# B&R Automation Studio project SuperTrakProject
Automation Studio 6.7.1.5

## Configuration APC4100

CPU 5APC4100.TGL1-000, AutomationRuntime 6.7.6, Build 11.3.0

### Task classes (Cpu.sw)
```
Cyclic#1 (cycle 800 us, tolerance 0 us):
  STCyclic <- Source.STMgr.STCyclic.STCyclic.prg
  STSystem <- Source.STMgr.STSystem.STSystem.prg
  STSection <- Source.STMgr.STSection.STSection.prg
  STTarget <- Source.STMgr.STTarget.STTarget.prg
  STShuttle <- Source.STMgr.STShuttle.STShuttle.prg
Cyclic#2 (cycle 1600 us, tolerance 1600 us):
  Main <- Source.MachineMgr.Main.prg
Cyclic#3 (cycle 20000 us, tolerance 20000 us):
  EipComm <- Source.EthIP.EipComm.prg
DataObjects: ethIPcon <- Source.EthIP.ethIPcon.dob
Binaries: udbdef, TCData, TCLang, ashwd, ashwac, sysconf, asfw, arconfig, TC, varmap, stcyclicvm
Libraries: ArEventLog, AsIOAcc, AsARCfg, AsArProf, AsArSdm, AsGuard, AsHttp, AsIO, AsIODiag, AsIOMMan, AsIoTime, AsTCP, astime, AsUDP, AsXml, brsystem, DataObj, FileIO, sys_lib, runtime, AsBrStr, standard, AsIecCon, AsEthIP, StCom, SuperTrak, ArTextSys, UserLog, aspciext
```

### Hardware
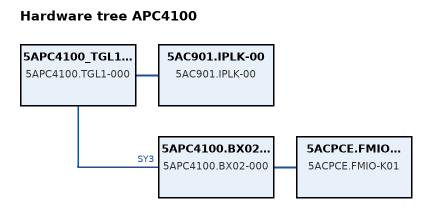
```
5AC901.IPLK-00 : 5AC901.IPLK-00 v2.1.0.0  [SS -> 5APC4100_TGL1_000.SS2]
  Connector IF1:
    CycleTime = 800
5ACPCE.FMIO-K01 : 5ACPCE.FMIO-K01 v1.0.6.0  [SL -> 5APC4100.BX02-000.SL1]
5APC4100.BX02-000 : 5APC4100.BX02-000 v1.0.0.0  [SY -> 5APC4100_TGL1_000.SY3]
5APC4100_TGL1_000 : 5APC4100.TGL1-000 v1.4.0.0
  Connector IF3:
    AssignedOperatingSystem = ARemb
    ActivateDevice = 1
    HostName = apc4100_supertrak
    Mode = Manual
    InternetAddress = 192.168.1.100
    SubnetMask = 255.255.255.0
    ActivateSnmp = 2
  Connector IF4:
    AssignedOperatingSystem = ARemb
    ActivateDevice = 1
    HostName = apc4100_supertrak
    Mode = Manual
    InternetAddress = 10.10.6.10
    SubnetMask = 255.255.255.0
    ActivateSnmp = 2
  Connector IF5:
    AssignedOperatingSystem = ARemb
    ActivateDevice = 1
    HostName = apc4100_supertrak
    ActivateSnmp = 2
  Connector IF6:
    AssignedOperatingSystem = ARemb
    ActivateDevice = 1
    HostName = apc4100_supertrak
    ActivateSnmp = 2
  Connector IF7:
    AssignedOperatingSystem = ARemb
  Connector IF8:
    AssignedOperatingSystem = ARemb
  Connector IF9:
    AssignedOperatingSystem = ARemb
  Connector IF10:
    AssignedOperatingSystem = ARemb
  Connector IF11:
    AssignedOperatingSystem = ARemb
  Connector IF12:
    AssignedOperatingSystem = ARemb
  ConfigurationID = SuperTrakProject_APC4100
  ConfigVersion = 2.0.0
  UserPartitionSize = 100
  EnableDebugger = 1
  TimerDeviceType = EPLX2X
  TimerDevice = 5AC901.IPLK-00.IF1
  TaskClassIdleTime = 800
  Cyclic1Duration = 800
  Cyclic1Tolerance = 0
  Cyclic2Duration = 1600
  Cyclic2Tolerance = 1600
  Cyclic3Duration = 20000
  Cyclic3Tolerance = 20000
  Cyclic8Duration = 9600
  FileDevice1
  FileDeviceName1 = USER
  FileDevicePath1 = USER_PATH
  EthernetHostName = apc4100_supertrak
  ActivateFtpServer = 1
  FtpUser1
  FtpUsername1 = SuperTrakUser
  FtpUserPassword1 = ss9kzLCmIlqrwmUb/fXl5DaWp4kAdzlsqUsPLdKHEtE=  // SuperTrak
  FtpUserSalt1 = yN37R9W0
  FTPAccessRight1 = 0
  ActivateWebServer = 1
  WebServerProtocol = 1
  ActivateSdm = 1
  Authentication = 0
```

## Configuration APC910

CPU 5APC4100.TGL1-000, AutomationRuntime 6.3.4, Build 11.3.0, Vc 6.0.0

CPU 5PC900.TS17-00, AutomationRuntime 6.3.4, Build 11.3.0, Vc 6.0.0

CPU 5PC900.TS77-00, AutomationRuntime G4.91, Build 4.1.2, Vc V4.72.5

### Task classes (Cpu.sw)
```
Cyclic#1 (cycle 800 us, tolerance 0 us):
  STCyclic <- Source.STMgr.STCyclic.STCyclic.prg
  STSystem <- Source.STMgr.STSystem.STSystem.prg [disabled]
  STSection <- Source.STMgr.STSection.STSection.prg [disabled]
  STTarget <- Source.STMgr.STTarget.STTarget.prg [disabled]
  STShuttle <- Source.STMgr.STShuttle.STShuttle.prg [disabled]
Cyclic#2 (cycle 1600 us, tolerance 1600 us):
  Main <- Source.MachineMgr.Main.prg [disabled]
Cyclic#4:
  EipComm <- Source.EthIP.EipComm.prg [disabled]
DataObjects: ethIPcon <- Source.EthIP.ethIPcon.dob
Binaries: STComTexts, udbdef, TCData, TCLang, ashwd, ashwac, sysconf, asfw, arconfig, TC, varmap, stcyclicvm
Libraries: SuperTrak, ArEventLog, AsIOAcc, AsARCfg, AsArLog, AsArProf, AsArSdm, AsGuard, AsHttp, AsIO, AsIODiag, AsIOMMan, AsIoTime, AsTCP, astime, AsUDP, AsXml, brsystem, DataObj, FileIO, sys_lib, runtime, StCom, AsBrStr, standard, AsIecCon, UserLog, AsEthIP, aspciext
```

### Task classes (Cpu.sw)
```
Cyclic#1 (cycle 800 us, tolerance 0 us):
  STCyclic <- Source.STMgr.STCyclic.STCyclic.prg
  STSystem <- Source.STMgr.STSystem.STSystem.prg
  STSection <- Source.STMgr.STSection.STSection.prg
  STTarget <- Source.STMgr.STTarget.STTarget.prg
  STShuttle <- Source.STMgr.STShuttle.STShuttle.prg
Cyclic#2 (cycle 1600 us, tolerance 1600 us):
  Main <- Source.MachineMgr.Main.prg
Cyclic#4:
  EipComm <- Source.EthIP.EipComm.prg
DataObjects: ethIPcon <- Source.EthIP.ethIPcon.dob
Binaries: STComTexts, udbdef, TCData, TCLang, ashwd, ashwac, sysconf, asfw, arconfig, TC, varmap, stcyclicvm
Libraries: SuperTrak, ArEventLog, AsIOAcc, AsARCfg, AsArLog, AsArProf, AsArSdm, AsGuard, AsHttp, AsIO, AsIODiag, AsIOMMan, AsIoTime, AsTCP, astime, AsUDP, AsXml, brsystem, DataObj, FileIO, sys_lib, runtime, StCom, AsBrStr, standard, AsIecCon, UserLog, AsEthIP, aspciext
```

### Hardware
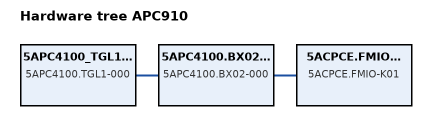
```
5ACPCE.FMIO-K01 : 5ACPCE.FMIO-K01 v1.0.6.0  [SL -> 5APC4100.BX02-000.SL1]
5APC4100.BX02-000 : 5APC4100.BX02-000 v1.0.0.0  [SY -> 5APC4100_TGL1_000.SY3]
5APC4100_TGL1_000 : 5APC4100.TGL1-000 v1.2.0.0
  Connector IF3:
    AssignedOperatingSystem = ARemb
    ActivateDevice = 1
    HostName = apc910_supertrak
    Mode = Manual
    InternetAddress = 192.168.1.100
    SubnetMask = 255.255.255.0
    ActivateSnmp = 2
  Connector IF4:
    AssignedOperatingSystem = ARemb
    ActivateDevice = 1
    HostName = apc910_supertrak
    Mode = Manual
    InternetAddress = 10.10.6.10
    SubnetMask = 255.255.255.0
    ActivateSnmp = 2
  Connector IF5:
    AssignedOperatingSystem = ARemb
    ActivateDevice = 1
  Connector IF6:
    AssignedOperatingSystem = ARemb
    ActivateDevice = 1
  Connector IF7:
    AssignedOperatingSystem = ARemb
  Connector IF8:
    AssignedOperatingSystem = ARemb
  Connector IF9:
    AssignedOperatingSystem = ARemb
  Connector IF10:
    AssignedOperatingSystem = ARemb
  Connector IF11:
    AssignedOperatingSystem = ARemb
  Connector IF12:
    AssignedOperatingSystem = ARemb
  ConfigurationID = SuperTrakProject_APC910
  ConfigVersion = 1.1.0
  UserPartitionSize = 100
  SystemTick = 800
  TaskClassIdleTime = 800
  Cyclic1Duration = 800
  Cyclic1Tolerance = 0
  Cyclic2Duration = 1600
  Cyclic2Tolerance = 1600
  Cyclic3Duration = 49600
  Cyclic3Tolerance = 49600
  Cyclic8Duration = 9600
  FileDevice1
  FileDeviceName1 = USER
  FileDevicePath1 = USER_PATH
  EthernetHostName = apc910_supertrak
  ActivateFtpServer = 1
  FtpUser1
  FtpUsername1 = SuperTrakUser
  FtpUserPassword1 = ss9kzLCmIlqrwmUb/fXl5DaWp4kAdzlsqUsPLdKHEtE=  // SuperTrak
  FtpUserSalt1 = yN37R9W0
  FTPAccessRight1 = 0
  ActivateWebServer = 1
  ActivateSdm = 1
```

### VarMap.vvm - 5PC900_TS17_00/VarMap.vvm
```iecst
VAR_CONFIG
	Cyclic#1.::gSTSection.Cmd AT %Q.Cyclic#1.::STSection:Interface.Cmd;
	Cyclic#1.::STSection:Interface.Status AT %Q.Cyclic#1.::gSTSection.Status;
END_VAR
```

### STCyclicVM.vvm - 5PC900_TS17_00/VariableMap/STCyclicVM.vvm
```iecst
VAR_CONFIG
	::STCyclic:Interface.Status AT %Q.::gSTCyclic.Status;
END_VAR
```

### STSystemVM.vvm - 5PC900_TS17_00/VariableMap/STSystemVM.vvm
```iecst
VAR_CONFIG
	::gSTSystem.Par AT %Q.::STSystem:Interface.Par;
END_VAR
```

### VarMap.vvm - 5PC900_TS77_00/VarMap.vvm
```iecst
VAR_CONFIG
	::gSTSystem.Cmd AT %Q.::STSystem:Interface.Cmd;
	::STSystem:Interface.Status AT %Q.::gSTSystem.Status;
	::gSTSection.Cmd AT %Q.::STSection:Interface.Cmd;
	::gSTSection.Par AT %Q.::STSection:Interface.Par;
	::STSection:Interface.Status AT %Q.::gSTSection.Status;
END_VAR
```

## Logical view

Binary libraries used (declarations not repeated): SuperTrak 0.63.4, StCom 6.0.0, brsystem, runtime, sys_lib, standard, astime, AsBrStr, AsIecCon, AsIOAcc, AsARCfg, AsArProf, AsArSdm, AsGuard, AsHttp, AsIO, AsIODiag, AsIOMMan, AsIoTime, AsTCP, AsUDP, AsXml, DataObj, FileIO, ArEventLog, UserLog 2.1.0, ArTextSys, AsEthIP

### Package Logical/Libraries - Global libraries

### Library Logical/Libraries/StHelper (IEC)
Depends on: SuperTrak, UserLog

#### Constants.var - Exported constants
```iecst
VAR CONSTANT
	ST_HELPER_FUNCTION_INPUT_ERROR : UINT := 20; (*Helper Function could not execute due to an invalid input*)
END_VAR
```

#### StHelper.fun - Exported functions and function blocks
```iecst
(*Data Parameters*)

FUNCTION GetDataParameterArrayLength : UINT (*Gets the array length for data parameters. The array length N indicates that N values can be addressed, using indexes 0 through (N - 1). Returned value is the Status of SuperTrakServChanRead*)
	VAR_INPUT
		ParameterToCheck : UINT; (*Data parameter number to check the length of*)
		pDataBuffer : UDINT; (*Pointer to (UDINT) location of output data*)
		DataBufferLength : UINT; (*[bytes] Size of output data location*)
	END_VAR
	VAR
		LogValues : UserLogFormatType; (*Runtime values formatted for Log messages*)
	END_VAR
END_FUNCTION
(*Inputs and Outputs*)

FUNCTION GetInputFunctions : UINT (*Gets the functions configured for all Trakmaster Inputs. Returned value is the Status of SuperTrakServChanRead*)
	VAR_INPUT
		pDataBuffer : UDINT; (*Pointer to (UINT[8]) location of output data. Each element in the array is a Digital Input.*)
		DataBufferLength : UINT; (*[bytes] Size of output data location*)
	END_VAR
	VAR
		GetArrayLengthStatus : UINT; (*Status returned by GetDataParameterArrayLength*)
		GetArrayLengthReturnValue : UDINT; (*Value returned by GetDataParameterArrayLength*)
		Count : UINT; (*Count of values to read*)
		LogValues : UserLogFormatType; (*Runtime values formatted for Log messages*)
	END_VAR
END_FUNCTION

FUNCTION SetInputFunctions : UINT (*Sets the functions configured for all Trakmaster Inputs. Returned value is the Status of SuperTrakServChanRead*)
	VAR_INPUT
		pDataBuffer : UDINT; (*Pointer to (UINT[8]) location of input data. Each element in the array is a Digital Input.*)
		DataBufferLength : UINT; (*[bytes] Size of input data location*)
	END_VAR
	VAR
		GetArrayLengthStatus : UINT; (*Status returned by GetDataParameterArrayLength*)
		GetArrayLengthReturnValue : UDINT; (*Value returned by GetDataParameterArrayLength*)
		Count : UINT; (*Count of values to read*)
		LogValues : UserLogFormatType; (*Runtime values formatted for Log messages*)
	END_VAR
END_FUNCTION
```

#### GetDataParameterArrayLength.st
```iecst
// Gets the array length for data parameters. The array length N indicates that N values can be addressed, using indexes 0 through (N - 1)
// An array length of 1 indicates that a single value can be addressed at index 0.
// An array length OF 0 indicates that the parameter is NOT available.
// Returned value is the Status of SuperTrakServChanRead
FUNCTION GetDataParameterArrayLength

    IF (ParameterToCheck < 1024) OR (pDataBuffer = 0) OR (DataBufferLength = 0) THEN
        GetDataParameterArrayLength := ST_HELPER_FUNCTION_INPUT_ERROR;
    ELSE
        // Data parameters occupy parameter numbers starting at 1024
        // To obtain information about data parameter K, specify index K - 1024 when reading the Data Parameter Information parameters
        GetDataParameterArrayLength := SuperTrakServChanRead(0, stPAR_PARAM_ARRAY_LENGTH, ParameterToCheck - 1024, 1, pDataBuffer, DataBufferLength);
        LogValues.i[0] := stPAR_PARAM_ARRAY_LENGTH;
        LogValues.i[1] := ParameterToCheck - 1024;
        LogValues.i[2] := 1;
        UserLogAdvanced(USERLOG_SEVERITY_INFORMATION, 100, 'Service Channel Request: Parameter %i, Start Index %i, Count %i', LogValues);
    END_IF;

END_FUNCTION
```

#### InputsAndOutputs.st
```iecst
// Gets the functions configured for all Trakmaster Inputs. Returned value is the Status of SuperTrakServChanRead
FUNCTION GetInputFunctions

    // Check inputs for validity
    IF (pDataBuffer = 0) OR (DataBufferLength = 0) THEN
        GetInputFunctions := ST_HELPER_FUNCTION_INPUT_ERROR;
        RETURN;
    END_IF;

    // Check size of data array
    GetArrayLengthStatus := GetDataParameterArrayLength(stPAR_DIGITAL_INPUT_FUNCTION, ADR(GetArrayLengthReturnValue), SIZEOF(GetArrayLengthReturnValue));
    IF GetArrayLengthStatus <> 0 THEN
        GetInputFunctions := ST_HELPER_FUNCTION_INPUT_ERROR;
        RETURN;
    END_IF;

    // Number of inputs is lesser of (data array size, size of data buffer elements)
    Count := MIN(UDINT_TO_UINT(GetArrayLengthReturnValue), DataBufferLength/SIZEOF(UINT));
    GetInputFunctions := SuperTrakServChanRead(0, stPAR_DIGITAL_INPUT_FUNCTION, 0, Count, pDataBuffer, DataBufferLength);
    LogValues.i[0] := stPAR_DIGITAL_INPUT_FUNCTION;
    LogValues.i[1] := 0;
    LogValues.i[2] := Count;
    UserLogAdvanced(USERLOG_SEVERITY_INFORMATION, 100, 'Service Channel Request: Parameter %i, Start Index %i, Count %i', LogValues);

END_FUNCTION

// Sets the functions configured for all Trakmaster Inputs. Returned value is the Status of SuperTrakServChanRead
FUNCTION SetInputFunctions

    // Check inputs for validity
    IF (pDataBuffer = 0) OR (DataBufferLength = 0) THEN
        SetInputFunctions := ST_HELPER_FUNCTION_INPUT_ERROR;
        RETURN;
    END_IF;

    // Check size of data array
    GetArrayLengthStatus := GetDataParameterArrayLength(stPAR_DIGITAL_INPUT_FUNCTION, ADR(GetArrayLengthReturnValue), SIZEOF(GetArrayLengthReturnValue));
    IF GetArrayLengthStatus <> 0 THEN
        SetInputFunctions := ST_HELPER_FUNCTION_INPUT_ERROR;
        RETURN;
    END_IF;

    // Number of inputs is lesser of (data array size, size of data buffer elements)
    Count := MIN(UDINT_TO_UINT(GetArrayLengthReturnValue), DataBufferLength/SIZEOF(UINT));
    SetInputFunctions := SuperTrakServChanWrite(0, stPAR_DIGITAL_INPUT_FUNCTION, 0, Count, pDataBuffer, DataBufferLength);
    LogValues.i[0] := stPAR_DIGITAL_INPUT_FUNCTION;
    LogValues.i[1] := 0;
    LogValues.i[2] := Count;
    UserLogAdvanced(USERLOG_SEVERITY_INFORMATION, 100, 'Service Channel Request: Parameter %i, Start Index %i, Count %i', LogValues);

END_FUNCTION
```

### Package Logical/Source/MachineMgr - Machine manager

### Machine.typ - Global Machine types
```iecst
(***************************************************************************************
 * Global Machine data types
 *
 * These structures allow any program (task) to interface with the Main Machine task
 *
 * File: Machine.typ
 * Created: 2024-08-15
 *
 * Authors:
 *  Marcus Mangel, B&R Industrial Automation
 *
****************************************************************************************)

TYPE
    Machine_type :     STRUCT  (*Machine interface*)
        Cmd : Machine_Cmd_type; (*Machine commands*)
        Par : Machine_Par_type; (*Machine parameters*)
        Status : Machine_Status_type; (*Machine statuses*)
    END_STRUCT;
    Machine_Cmd_type :     STRUCT  (*Machine commands*)
        Power : BOOL; (*Power all SuperTrak sections*)
        Run : BOOL; (*Run process sequence*)
        ErrorReset : BOOL; (*Error reset*)
    END_STRUCT;
    Machine_Par_type :     STRUCT  (*Machine parameters*)
        Velocity : REAL := 1500.0; (*[mm/s] Set velocity for target and shuttle release commands*)
        Acceleration : REAL := 15.0; (*[m/s^2] Set acceleration for target and shuttle release commands*)
    END_STRUCT;
    Machine_Status_type :     STRUCT  (*Machine statuses*)
        PowerOn : BOOL; (*The main state machine is enabled and the trak is powered*)
        Ready : BOOL; (*The program is ready to run*)
        Error : BOOL; (*There is an active error present*)
        ErrorType : Error_Type_enum; (*Source of the last error*)
        ErrorText : STRING[255];
        SuperTrakDiag : SuperTrak_Diag_type; (*Fault and Warning information from the SuperTrak library*)
    END_STRUCT;
    Error_Type_enum :
        ( (*Source of the last error*)
        errNONE := 0,
        errUSER := 1, (*See Automation Studio code*)
        errST_COM_SYSTEM := 2, (*See documentation for the StCom or SuperTrak libraries in Automation Studio*)
        errST_COM_SECTION := 3, (*See documentation for the StCom or SuperTrak libraries in Automation Studio*)
        errST_SYSTEM := 10, (*See "Faults" section in TrakMaster Help *)
        warnST_SYSTEM := 11, (*See "Warnings" section in TrakMaster Help *)
        errST_SECTION := 20, (*See "Faults" section in TrakMaster Help *)
        warnST_SECTION := 21, (*See "Warnings" section in TrakMaster Help *)
        errST_COM_TARGET := 30, (*See documentation for the StCom or SuperTrak libraries in Automation Studio*)
        errST_COM_SHUTTLE := 40 (*See documentation for the StCom or SuperTrak libraries in Automation Studio*)
        );
    SuperTrak_Diag_type :     STRUCT  (*Fault and Warning information from the SuperTrak library*)
        SuperTrakDiagIndex : USINT; (*Index 0 is the System, others are for a specific section. Set to a relevant index when Errors occur*)
        Warnings : ARRAY[0..31]OF BOOL; (*See TrakMaster Help for descriptions*)
        Errors : ARRAY[0..31]OF BOOL; (*See TrakMaster Help for descriptions*)
    END_STRUCT;
END_TYPE
```

### Machine.var - Global Machine variables
```iecst
(***************************************************************************************
 * Global Machine variables
 *
 * These variables allow any program (task) to interface with the Main Machine task
 *
 * File: Machine.var
 * Created: 2024-08-15
 *
 * Authors:
 *  Marcus Mangel, B&R Industrial Automation
 *
***************************************************************************************)
VAR
    gMachine : Machine_type; (*Machine interface*)
    gUseExternalControl : BOOL;
END_VAR
```

### Program Logical/Source/MachineMgr/Main (IEC) - Main Machine control

#### Main.st - Init, cyclic, exit code
```iecst
(***************************************************************************************
 * Main task
 *
 * This task (program) provides a state machine for controlling any and all hardware
 * connected to the B&R PC. SuperTrak (Target) release code is demonstrated in the
 * MAIN_STATE_RUN (Running) state of this state machine.
 *
 * Other tasks can interface with this one via the global variable "gMachine".
 *
 * File: Main.st
 * Created: 2024-08-15
 *
 * Authors:
 *  Marcus Mangel, B&R Industrial Automation
 *  Bryan Olson, B&R Industrial Automation
 *
***************************************************************************************)

PROGRAM _INIT

    // Set simulated station timer values
    SimulatedProcessTimes[ST_TARGET_LOAD] := T#1s;
    SimulatedProcessTimes[ST_TARGET_QUEUE] := T#100ms;
    SimulatedProcessTimes[ST_TARGET_PROCESS] := T#500ms;
    SimulatedProcessTimes[ST_TARGET_UNLOAD] := T#1s;

END_PROGRAM

PROGRAM _CYCLIC

    // Copy inputs
    Interface.Cmd := gMachine.Cmd;
    Interface.Par := gMachine.Par;

    // Check for command edges
    r_trig_Power(CLK := Interface.Cmd.Power);
    r_trig_Run(CLK := Interface.Cmd.Run);

    // Translate Errors
    GetErrorType;
    GetTrakMasterWarningsAndErrors;
    // Catch SuperTrak Errors
    IF gSuperTrak.System.Status.Error OR gSuperTrak.System.Info.FaultPresent
        OR gSuperTrak.Sections.Status.Error OR (gSuperTrak.Sections.Status.SectionError <> 0)
        OR TargetErrorPresent OR ShuttleErrorPresent THEN

        IF gSuperTrak.System.Info.FaultPresent THEN
            Interface.Status.SuperTrakDiag.SuperTrakDiagIndex:= 0;
        ELSE
            FOR i:= 1 TO SIZEOF(gSuperTrak.Sections.Info)/SIZEOF(gSuperTrak.Sections.Info[1]) DO
                IF gSuperTrak.Sections.Info[i].FaultPresent THEN
                    Interface.Status.SuperTrakDiag.SuperTrakDiagIndex:= i;
                    EXIT;
                END_IF
            END_FOR
        END_IF

        // Then go to Error State
        MainState := MAIN_STATE_ERROR;

    END_IF;
    // Reset Errors
    gSuperTrak.System.Cmd.Reset := Interface.Cmd.ErrorReset;

    // Disable handling
    // Go to the Disabled state whenever gSuperTrak.System.Status.Active drops
    // Only respond to Interface.Command.Power if gUseExternalControl is false
    IF ((NOT gUseExternalControl AND NOT Interface.Cmd.Power) OR NOT gSuperTrak.System.Status.Active)
        AND (MainState > MAIN_STATE_DISABLED) AND (MainState < MAIN_STATE_DISABLING) THEN
        MainState := MAIN_STATE_DISABLING;
    END_IF;

    // Main State Machine
    // State machine is passive if main logic is external
    // States will reflect overall machine status, but will not
    // control the SuperTrak
    CASE MainState OF
        MAIN_STATE_OFF:
            IF NOT gUseExternalControl THEN
                gSuperTrak.System.Cmd.PowerAllSections := FALSE;
            END_IF;

            // Wait for System and Sections to be Active
            IF gSuperTrak.System.Status.Active AND gSuperTrak.Sections.Status.Active THEN
                MainState := MAIN_STATE_DISABLED;
            END_IF;

        MAIN_STATE_DISABLED:
            // Reset commands and timers
            IF NOT gUseExternalControl THEN
                ResetTargetRelease;
                ResetShuttleRelease;
                ResetProcessTimer;
            END_IF;

            IF r_trig_Power.Q AND gSuperTrak.System.Status.Ready AND NOT gUseExternalControl THEN
                MainState := MAIN_STATE_POWER_SECTIONS;
            ELSIF gUseExternalControl AND gSuperTrak.System.Info.SectionsEnabled THEN
                MainState := MAIN_STATE_READY; // Power and Recovery steps should be handled externally
            END_IF;

        MAIN_STATE_POWER_SECTIONS:
            IF NOT gUseExternalControl THEN
                gSuperTrak.System.Cmd.PowerAllSections := TRUE;
            END_IF;

            IF gSuperTrak.System.Info.SectionsEnabled THEN
                MainState := MAIN_STATE_RECOVER;
            END_IF;

        MAIN_STATE_RECOVER:
            GetTargetsReleased;
            GetShuttlesReleased;
            IF TargetsReleased AND ShuttlesReleased AND gSuperTrak.System.Status.PowerOn THEN // Recovered and at standstill
                // Add conditions to satisfy process recovery
                MainState := MAIN_STATE_READY;
            END_IF

        MAIN_STATE_READY:
            IF r_trig_Run.Q AND NOT gUseExternalControl THEN
                MainState := MAIN_STATE_RUN;
            END_IF;

        MAIN_STATE_RUN:
            IF gUseExternalControl OR NOT Interface.Cmd.Run THEN
                MainState := MAIN_STATE_READY;
            ELSE
                MainLogic; // Target release code goes in this Action
            END_IF

        MAIN_STATE_DISABLING:
            IF NOT gUseExternalControl THEN
                gSuperTrak.System.Cmd.PowerAllSections := FALSE;
            END_IF;

            IF gSuperTrak.System.Info.SectionsDisabled THEN
                MainState := MAIN_STATE_DISABLED;
            END_IF;

        MAIN_STATE_ERROR:
            IF NOT gUseExternalControl THEN
                gSuperTrak.System.Cmd.PowerAllSections := FALSE;

                // Reset commands and timers
                ResetTargetRelease;
                ResetShuttleRelease;
                ResetProcessTimer;
            END_IF;

            IF Interface.Cmd.ErrorReset
                AND NOT gSuperTrak.System.Status.Error AND (gSuperTrak.Sections.Status.SectionError = 0)
                AND NOT TargetErrorPresent AND NOT ShuttleErrorPresent THEN
                MainState := MAIN_STATE_OFF;
            END_IF;
    END_CASE;

    // Call function blocks
    fb_ArTextSysGetText.Namespace := ADR('User/SuperTrakErrors');
    fb_ArTextSysGetText.LanguageCode := 'en';
    fb_ArTextSysGetText.TextBuffer := ADR(Interface.Status.ErrorText);
    fb_ArTextSysGetText.TextBufferSize := SIZEOF(Interface.Status.ErrorText);
    fb_ArTextSysGetText();
    IF fb_ArTextSysGetText.Done THEN
        fb_ArTextSysGetText.Execute := FALSE;
    END_IF;

    // Set statuses
    Interface.Status.PowerOn := ((Interface.Cmd.Power) AND (MainState > MAIN_STATE_DISABLED));
    Interface.Status.Ready := (MainState = MAIN_STATE_READY);
    Interface.Status.Error := (MainState = MAIN_STATE_ERROR);

    // Copy outputs
    gMachine.Status := Interface.Status;

END_PROGRAM
```

#### Types.typ - Local data types
```iecst
(***************************************************************************************
 * Main task local data types
 *
 * These structures and enumerations are local to the Main task
 *
 * File: Main/Types.typ
 * Created: 2024-08-15
 *
 * Authors:
 *  Marcus Mangel, B&R Industrial Automation
 *
***************************************************************************************)

TYPE
	MainState_enum :
		( (*Program state*)
		MAIN_STATE_OFF, (*SuperTrak control is disabled*)
		MAIN_STATE_DISABLED, (*SuperTrak control is enabled, but the trak itself is disabled*)
		MAIN_STATE_POWER_SECTIONS, (*SuperTrak sections are enabling and powering up*)
		MAIN_STATE_RECOVER, (*Shuttles are recovering*)
		MAIN_STATE_READY, (*Trak is ready to run the main process*)
		MAIN_STATE_RUN, (*Trak is running the main process*)
		MAIN_STATE_DISABLING, (*Trak is disabling all sections*)
		MAIN_STATE_ERROR (*There is an active error*)
		);
END_TYPE
```

#### Variables.var - Local variables
```iecst
(***************************************************************************************
 * Main task local variables
 *
 * These variables are local to the Main task
 *
 * File: Main/Variables.var
 * Created: 2024-08-15
 *
 * Authors:
 *  Marcus Mangel, B&R Industrial Automation
 *
***************************************************************************************)
(*Control*)
VAR
    MainState : MainState_enum; (*Program state*)
    Interface : Machine_type; (*Local copy of gMachine*)
    SimulatedProcessTimes : ARRAY[1..ST_TARGET_MAX] OF TIME; (*Times used to simulate machine processes*)
    LoopTarget : USINT; (*FOR loop index*)
    LoopShuttle : USINT; (*FOR loop index*)
    TextID : STRING[80];
    TargetErrorPresent : BOOL;
    ShuttleErrorPresent : BOOL;
    i : USINT;
END_VAR
(*Status*)
VAR
    TargetsReleased : BOOL; (*All configured target release commands confirmed*)
    ShuttlesReleased : BOOL; (*All configured shuttle release commands confirmed*)
END_VAR
(*Function Blocks*)
VAR
    ProcessTimer : ARRAY[1..ST_TARGET_MAX] OF TON; (*Timers used to simulate machine processes*)
    r_trig_Power : R_TRIG; (*Rising edge checker for Power command*)
    r_trig_Run : R_TRIG; (*Rising edge checker for Run command*)
    fb_ArTextSysGetText : ArTextSysGetText; (*Get error texts*)
END_VAR
(*Constants*)
VAR CONSTANT
    ST_TARGET_LOAD : USINT := 1;
    ST_TARGET_QUEUE : USINT := 2;
    ST_TARGET_PROCESS : USINT := 3;
    ST_TARGET_UNLOAD : USINT := 4;
END_VAR
```

#### MainLogic.st - Main state machine
```iecst
(***************************************************************************************
 * Main State Machine
 *
 * This Action should be placed in the RUN state of the Main State Machine.
 * It interfaces with the gSuperTrak structure to read statuses and write back
 * shuttle release commands.
 *
 * If the main machine logic is written elsewhere (e.g., in an AB PLC), this Action
 * should not be run. Instead, data is passed to/from gSuperTrak via the EipComm task.
 *
 * File: Main/MainLogic.st
 * Created: 2026-06-19
 *
 * Authors:
 *  Marcus Mangel, B&R Industrial Automation
 *
***************************************************************************************)

ACTION MainLogic:

    (*******************************************************
     *******************************************************
                Target control code goes here
    *******************************************************
    *******************************************************)

    // In simulation, timers are used to simulate process stations
    // On a real system, release commands should come from a real signal (e.g., a Digital Input)
    FOR LoopTarget := 1 TO ST_TARGET_MAX DO
        ProcessTimer[LoopTarget].IN := gSuperTrak.Target[LoopTarget].Status.ShuttlePresent;
        ProcessTimer[LoopTarget].PT := SimulatedProcessTimes[LoopTarget];
        ProcessTimer[LoopTarget]();
    END_FOR;

    // Target 1: Load
    IF ProcessTimer[ST_TARGET_LOAD].Q THEN
        IF gSuperTrak.Target[ST_TARGET_LOAD].Cmd.Release.ReleaseToTarget = FALSE THEN // Rising edge (one-shot)
            gSuperTrak.Target[ST_TARGET_LOAD].Par.Release.Velocity := Interface.Par.Velocity;
            gSuperTrak.Target[ST_TARGET_LOAD].Par.Release.Acceleration := Interface.Par.Acceleration;
            gSuperTrak.Target[ST_TARGET_LOAD].Par.Release.Direction := gSuperTrak.System.Par.GlobalDirection;
            gSuperTrak.Target[ST_TARGET_LOAD].Par.Release.DestinationTarget := ST_TARGET_QUEUE;
            gSuperTrak.Target[ST_TARGET_LOAD].Cmd.Release.ReleaseToTarget := TRUE;
        END_IF
    END_IF

    // Target 2: Queue
    IF ProcessTimer[ST_TARGET_QUEUE].Q AND gSuperTrak.Target[ST_TARGET_PROCESS].Status.ShuttleCount = 0 THEN
        IF gSuperTrak.Target[ST_TARGET_QUEUE].Cmd.Release.ReleaseToTarget = FALSE THEN // Rising edge (one-shot)
            gSuperTrak.Target[ST_TARGET_QUEUE].Par.Release.Velocity := Interface.Par.Velocity;
            gSuperTrak.Target[ST_TARGET_QUEUE].Par.Release.Acceleration := Interface.Par.Acceleration;
            gSuperTrak.Target[ST_TARGET_QUEUE].Par.Release.Direction := gSuperTrak.System.Par.GlobalDirection;
            gSuperTrak.Target[ST_TARGET_QUEUE].Par.Release.DestinationTarget := ST_TARGET_PROCESS;
            gSuperTrak.Target[ST_TARGET_QUEUE].Cmd.Release.ReleaseToTarget := TRUE;
        END_IF
    END_IF

    // Target 3: Process
    IF ProcessTimer[ST_TARGET_PROCESS].Q THEN
        IF gSuperTrak.Target[ST_TARGET_PROCESS].Cmd.Release.ReleaseToTarget = FALSE THEN // Rising edge (one-shot)
            gSuperTrak.Target[ST_TARGET_PROCESS].Par.Release.Velocity := Interface.Par.Velocity;
            gSuperTrak.Target[ST_TARGET_PROCESS].Par.Release.Acceleration := Interface.Par.Acceleration;
            gSuperTrak.Target[ST_TARGET_PROCESS].Par.Release.Direction := gSuperTrak.System.Par.GlobalDirection;
            gSuperTrak.Target[ST_TARGET_PROCESS].Par.Release.DestinationTarget := ST_TARGET_UNLOAD;
            gSuperTrak.Target[ST_TARGET_PROCESS].Cmd.Release.ReleaseToTarget := TRUE;
        END_IF
    END_IF

    // Target 4: Unload
    IF ProcessTimer[ST_TARGET_UNLOAD].Q THEN
        IF gSuperTrak.Target[ST_TARGET_UNLOAD].Cmd.Release.ReleaseToTarget = FALSE THEN // Rising edge (one-shot)
            gSuperTrak.Target[ST_TARGET_UNLOAD].Par.Release.Velocity := Interface.Par.Velocity;
            gSuperTrak.Target[ST_TARGET_UNLOAD].Par.Release.Acceleration := Interface.Par.Acceleration;
            gSuperTrak.Target[ST_TARGET_UNLOAD].Par.Release.Direction := gSuperTrak.System.Par.GlobalDirection;
            gSuperTrak.Target[ST_TARGET_UNLOAD].Par.Release.DestinationTarget := ST_TARGET_LOAD;
            gSuperTrak.Target[ST_TARGET_UNLOAD].Cmd.Release.ReleaseToTarget := TRUE;
        END_IF
    END_IF

    // Reset commands
    FOR LoopTarget := 1 TO ST_TARGET_MAX DO
        IF gSuperTrak.Target[LoopTarget].Status.ShuttleReleased THEN
            brsmemset(ADR(gSuperTrak.Target[LoopTarget].Cmd), 0, SIZEOF(gSuperTrak.Target[LoopTarget].Cmd));
        END_IF
    END_FOR

END_ACTION
```

#### Subroutines.st - Helper actions
```iecst
(***************************************************************************************
 * Main task subroutines (Actions)
 *
 * These Actions can be run only by the Main task
 *
 * File: Main/Subroutines.st
 * Created: 2024-08-15
 *
 * Authors:
 *  Marcus Mangel, B&R Industrial Automation
 *  Bryan Olson, B&R Industrial Automation
 *
***************************************************************************************)

(* Determine cummulative target released status *)
ACTION GetTargetsReleased:

    TargetsReleased := TRUE; // Assume true
    FOR LoopTarget := 1 TO ST_TARGET_MAX DO
        // Configured targets
        IF gSuperTrak.Target[LoopTarget].Status.Section <> 0 THEN
            // Any target command true while released confirmation false
            IF (gSuperTrak.Target[LoopTarget].Cmd.Release.ReleaseToTarget
                OR gSuperTrak.Target[LoopTarget].Cmd.Release.ReleaseToOffset
                OR gSuperTrak.Target[LoopTarget].Cmd.Release.IncrementOffset)
                AND NOT gSuperTrak.Target[LoopTarget].Status.ShuttleReleased THEN
                TargetsReleased := FALSE; // Disqualify
                EXIT;
            END_IF
        END_IF
    END_FOR

END_ACTION

(* Determine cummulative pallet released status *)
ACTION GetShuttlesReleased:

    ShuttlesReleased := TRUE; // Assume true
    FOR LoopShuttle := 1 TO ST_SHUTTLE_MAX DO
        // Pallet present on system
        IF gSuperTrak.Shuttle[LoopShuttle].Status.Present THEN
            // Any pallet command true while released confirmation false
            IF (gSuperTrak.Shuttle[LoopShuttle].Cmd.ReleaseToTarget
                OR gSuperTrak.Shuttle[LoopShuttle].Cmd.ReleaseToOffset
                OR gSuperTrak.Shuttle[LoopShuttle].Cmd.IncrementOffset)
                AND NOT gSuperTrak.Shuttle[LoopShuttle].Status.ShuttleReleased THEN
                ShuttlesReleased := FALSE; // Disqualify
                EXIT;
            END_IF
        END_IF
    END_FOR

END_ACTION

(* Reset all target release commands *)
ACTION ResetTargetRelease:

    FOR LoopTarget := 1 TO ST_TARGET_MAX DO
        brsmemset(ADR(gSuperTrak.Target[LoopTarget].Cmd), 0, SIZEOF(gSuperTrak.Target[LoopTarget].Cmd));
    END_FOR

END_ACTION

(* Reset all shuttle release commands *)
ACTION ResetShuttleRelease:

    FOR LoopShuttle := 1 TO ST_SHUTTLE_MAX DO
        brsmemset(ADR(gSuperTrak.Shuttle[LoopShuttle].Cmd), 0, SIZEOF(gSuperTrak.Shuttle[LoopShuttle].Cmd));
    END_FOR

END_ACTION

(* Reset all process timers *)
ACTION ResetProcessTimer:

    FOR LoopTarget := 1 TO ST_TARGET_MAX DO
        ProcessTimer[LoopTarget](IN := FALSE);
    END_FOR

END_ACTION

(* Set ErrorType depending on what caused the error *)
ACTION GetErrorType:

	// Clear ErrorType
    IF Interface.Cmd.ErrorReset OR MainState <> MAIN_STATE_ERROR THEN
        Interface.Status.ErrorType:= errNONE;
        brsmemset(ADR(Interface.Status.ErrorText), 0, SIZEOF(Interface.Status.ErrorText));
    END_IF

    // Default to User Error
    IF MainState = MAIN_STATE_ERROR AND Interface.Status.ErrorType = errNONE THEN
        Interface.Status.ErrorType:= errUSER;
    END_IF
    // System FUB Errors
    IF gSuperTrak.System.Status.Error THEN
        MainState:= MAIN_STATE_ERROR;
        Interface.Status.ErrorType:= errST_COM_SYSTEM;
        TextID := DINT_TO_STRING(gSuperTrak.System.Status.ErrorID);
        fb_ArTextSysGetText.TextID := ADR(TextID);
        fb_ArTextSysGetText.Execute := TRUE; // Set false after function block call
    END_IF
    // Section FUB Errors
    IF gSuperTrak.Sections.Status.Error THEN
        MainState:= MAIN_STATE_ERROR;
        Interface.Status.ErrorType:= errST_COM_SECTION;
        TextID := DINT_TO_STRING(gSuperTrak.Sections.Status.StatusID);
        fb_ArTextSysGetText.TextID := ADR(TextID);
        fb_ArTextSysGetText.Execute := TRUE; // Set false after function block call
    END_IF
    // System Warnings
    IF gSuperTrak.System.Info.WarningPresent THEN
        Interface.Status.ErrorType:= warnST_SYSTEM;
    END_IF
    // System Errors
    IF gSuperTrak.System.Info.FaultPresent THEN
        MainState:= MAIN_STATE_ERROR;
        Interface.Status.ErrorType:= errST_SYSTEM;
    END_IF
    // Section Warnings
    IF gSuperTrak.Sections.Status.SectionWarning <> 0 THEN
        Interface.Status.ErrorType:= warnST_SECTION;
    END_IF
    // Section Errors
    IF gSuperTrak.Sections.Status.SectionError <> 0 THEN
        MainState:= MAIN_STATE_ERROR;
        Interface.Status.ErrorType:= errST_SECTION;
    END_IF
    // Target Errors
    TargetErrorPresent := FALSE;
    FOR LoopTarget := 1 TO ST_TARGET_MAX DO
        IF gSuperTrak.Target[LoopTarget].Status.Error THEN
            MainState:= MAIN_STATE_ERROR;
            TargetErrorPresent := TRUE;
            Interface.Status.ErrorType:= errST_COM_TARGET;
            TextID := DINT_TO_STRING(gSuperTrak.Target[LoopTarget].Status.StatusID);
            fb_ArTextSysGetText.TextID := ADR(TextID);
            fb_ArTextSysGetText.Execute := TRUE; // Set false after function block call
        END_IF
    END_FOR
    // Shuttle Errors
    ShuttleErrorPresent := FALSE;
    FOR LoopShuttle := 1 TO ST_SHUTTLE_MAX DO
        IF gSuperTrak.Shuttle[LoopShuttle].Status.Error THEN
            MainState:= MAIN_STATE_ERROR;
            ShuttleErrorPresent := TRUE;
            Interface.Status.ErrorType:= errST_COM_SHUTTLE;
            TextID := DINT_TO_STRING(gSuperTrak.Shuttle[LoopShuttle].Status.StatusID);
            fb_ArTextSysGetText.TextID := ADR(TextID);
            fb_ArTextSysGetText.Execute := TRUE; // Set false after function block call
        END_IF
    END_FOR

END_ACTION

(* Translate bit-packed Errors and Warnings into Booleans *)
ACTION GetTrakMasterWarningsAndErrors:

    IF Interface.Status.SuperTrakDiag.SuperTrakDiagIndex = 0 THEN
        // System
        FOR i := 0 TO 31 DO
            Interface.Status.SuperTrakDiag.Warnings[i]	:= BIT_TST(gSuperTrak.System.Info.Warnings, i);
            Interface.Status.SuperTrakDiag.Errors[i] 	:= BIT_TST(gSuperTrak.System.Info.Faults, i);
        END_FOR
    ELSE
        // Sections
        FOR i := 0 TO 31 DO
            Interface.Status.SuperTrakDiag.Warnings[i]	:= BIT_TST(gSuperTrak.Sections.Info[Interface.Status.SuperTrakDiag.SuperTrakDiagIndex].Warnings, i);
            Interface.Status.SuperTrakDiag.Errors[i] 	:= BIT_TST(gSuperTrak.Sections.Info[Interface.Status.SuperTrakDiag.SuperTrakDiagIndex].Faults, i);
        END_FOR
    END_IF

END_ACTION
```

### STCyclic.typ
```iecst
TYPE
	STCyclicReferenceType : 	STRUCT
		ControlDataAddress : UDINT;
		ControlDataSize : UDINT;
		StatusDataAddress : UDINT;
		StatusDataSize : UDINT;
		RequestDataAddress : UDINT;
		RequestDataSize : UDINT;
		ResponseDataAddress : UDINT;
		ResponseDataSize : UDINT;
	END_STRUCT;
END_TYPE
```

### Machine.typ
```iecst
TYPE
	Machine_type : 	STRUCT
		Cmd : Machine_Cmd_type;
		Status : Machine_Status_type;
	END_STRUCT;
	Machine_Cmd_type : 	STRUCT
		Enable : BOOL;
		Run : BOOL;
	END_STRUCT;
	Machine_Status_type : 	STRUCT
		Error : BOOL;
	END_STRUCT;
END_TYPE
```

### Program Logical/Source/MachineMgr/STMgr/Main (IEC)

#### Types.typ
```iecst
TYPE
	MainState_enum :
		(
		MAIN_STATE_OFF,
		MAIN_STATE_INITIALIZE,
		MAIN_STATE_IDLE,
		MAIN_STATE_ENABLE_SECTIONS,
		MAIN_STATE_RUNNING,
		MAIN_STATE_STOPPING,
		MAIN_STATE_ERROR,
		MAIN_STATE_RESET
		);
END_TYPE
```

#### Variables.var
```iecst
VAR
	MainState : MainState_enum;
	Interface : Machine_type;
	LoopSection : USINT;
	AllSectionsEnabled : BOOL;
	EnableTrigger : R_TRIG;
	RunTrigger : R_TRIG;
END_VAR
```

#### Main.st
```iecst
PROGRAM _INIT
	(* Insert code here *)

END_PROGRAM

PROGRAM _CYCLIC

    // Copy commands
    Interface.Cmd := gMachine.Cmd;

    // Edge triggers
    EnableTrigger(CLK := Interface.Cmd.Enable);
    RunTrigger(CLK := Interface.Cmd.Run);

    // Error Handling
    IF gSTSystem.Status.Error OR gSTSection.Status.Error THEN
        MainState := MAIN_STATE_ERROR;
    END_IF;

    // Main state machine
    CASE MainState OF
        MAIN_STATE_OFF:
            IF EnableTrigger.Q THEN
                gSTSystem.Cmd.Enable := TRUE;
            END_IF;

            IF gSTSystem.Status.Active THEN
                MainState := MAIN_STATE_INITIALIZE;
            END_IF;

        MAIN_STATE_INITIALIZE:
            gSTSection.Cmd.Enable := TRUE;

            IF gSTSection.Status.Active THEN
                MainState := MAIN_STATE_IDLE;
            END_IF;

        MAIN_STATE_IDLE:
            IF RunTrigger.Q THEN
                MainState := MAIN_STATE_ENABLE_SECTIONS;
            END_IF;

        MAIN_STATE_ENABLE_SECTIONS:
            AllSectionsEnabled := TRUE; // Set True now, set False later if any section isn't ready
            FOR LoopSection := 1 TO ST_SECTION_MAX DO
                gSTSection.Cmd.EnableSection[LoopSection] := TRUE;
                IF NOT gSTSection.Status.SectionEnabled[LoopSection] THEN
                    AllSectionsEnabled := FALSE;
                END_IF;
            END_FOR;

            IF AllSectionsEnabled THEN
                MainState := MAIN_STATE_RUNNING;
            END_IF;

        MAIN_STATE_RUNNING:
            IF NOT Interface.Cmd.Run THEN
                MainState := MAIN_STATE_STOPPING;
            END_IF;

        MAIN_STATE_STOPPING:

        MAIN_STATE_ERROR:
            gSTSystem.Cmd.Enable := FALSE;
            gSTSystem.Cmd.Run := FALSE;

            gSTSection.Cmd.Enable := FALSE;
            FOR LoopSection := 1 TO ST_SECTION_MAX DO
                gSTSection.Cmd.EnableSection[LoopSection] := FALSE;
            END_FOR;
    END_CASE;

    // Copy statuses
    gMachine.Status := Interface.Status;

END_PROGRAM

PROGRAM _EXIT
	(* Insert code here *)

END_PROGRAM
```

### Package Logical/Source/MachineMgr/STMgr/STCyclic - SuperTrak cyclic update

### STCyclic.typ - Global types
```iecst
TYPE
	STCyclicRefType : 	STRUCT
		ControlDataAddress : UDINT;
		ControlDataSize : UDINT;
		StatusDataAddress : UDINT;
		StatusDataSize : UDINT;
		RequestDataAddress : UDINT;
		RequestDataSize : UDINT;
		ResponseDataAddress : UDINT;
		ResponseDataSize : UDINT;
	END_STRUCT;
END_TYPE
```

### STCyclic.var - Global variables
```iecst
VAR
	gSTCyclicRef : STCyclicRefType;
END_VAR
```

### Program Logical/Source/MachineMgr/STMgr/STCyclic/STCyclic (IEC) - SuperTrak cyclic update

#### Main.st - Init, cyclic, exit code
```iecst
PROGRAM _INIT

	// Initialize SuperTrak, set configuration path
	SuperTrakInit('/DEVICE=USER_PATH\SuperTrak\Configuration', '127.0.0.1', 'IF3,IF4');

	InitializeControlInterface;
	InitializeServiceChannel;

END_PROGRAM

PROGRAM _CYCLIC

	// Data addresses for PLC control interface
	AddressControlInterface;

	// StCom input data
	SuperTrakProcessControl(0, InterfaceParameters);

	// SuperTrak cyclic update
	SuperTrakCyclic1();

	// StCom output data
	SuperTrakProcessStatus(0, InterfaceParameters);

	// StCom configuration
	ProcessServiceChannel;

	// StCom reference
	ReferenceCyclicData;

END_PROGRAM

PROGRAM _EXIT

	SuperTrakExit();

END_PROGRAM
```

#### Interface.var - Control interface variables for PLC communication
```iecst
VAR
	ControlInterfaceRevision : UINT; (*Revision number 0 required for StCom*)
	ControlData : ARRAY[0..499] OF USINT; (*Raw input data to control interface*)
	StatusData : ARRAY[0..499] OF USINT; (*Raw output data from control interface*)
	InterfaceParameters : SuperTrakControlInterface_t; (*Control interface parameters*)
END_VAR
```

#### Interface.st - Control interface actions for PLC communication
```iecst
(* Assign revision, connection type, and size of control interface data *)
ACTION InitializeControlInterface:

	// Revision 0 required by StCom
	ControlInterfaceRevision := 0;
	SuperTrakServChanWrite(0, stPAR_PLC_IF_REVISION, 0, 1,
		ADR(ControlInterfaceRevision), SIZEOF(ControlInterfaceRevision));

	// Parameters used in SuperTrak ProcessControl and ProcessStatus functions
	InterfaceParameters.connectionType := stCONNECTION_LOCAL;
	InterfaceParameters.controlSize := SIZEOF(ControlData);
	InterfaceParameters.statusSize := SIZEOF(StatusData);

END_ACTION

(* Assign addresses of control interface data *)
ACTION AddressControlInterface:

	// Parameters used in SuperTrak ProcessControl and ProcessStatus functions
	InterfaceParameters.pControl := ADR(ControlData);
	InterfaceParameters.pStatus := ADR(StatusData);

END_ACTION
```

#### Service.var - Service channel variables
```iecst
VAR
	RequestData : ARRAY[0..127] OF USINT; (*Raw service channel input data*)
	ResponseData : ARRAY[0..127] OF USINT; (*Raw service channel output data*)
	ServiceChannel : ServiceChannel_t; (*Service channel instance interface*)
	RequestHeader : REFERENCE TO ServiceChannelHeader_t; (*Pointer to header in service channel input*)
	ResponseHeader : REFERENCE TO ServiceChannelHeader_t; (*Pointer to header in sercive channel output*)
	Values : UserLogFormatType; (*Runtime values for formatted log messages*)
END_VAR
```

#### Service.st - Service channel actions
```iecst
(* Assign channel ID and size of service channel data *)
ACTION InitializeServiceChannel:

	ServiceChannel.channelId := 1;

	ServiceChannel.requestBufferSize := SIZEOF(RequestData) - SIZEOF(ServiceChannelHeader_t);
	ServiceChannel.responseBufferSize := SIZEOF(ResponseData) - SIZEOF(ServiceChannelHeader_t);

END_ACTION

(* Assign addresses of service channel data *)
ACTION AddressServiceChannel:

	ServiceChannel.pRequestHeader := ADR(RequestData);
	ServiceChannel.pResponseHeader := ADR(ResponseData);
	ServiceChannel.pRequestValues := ADR(RequestData) + SIZEOF(ServiceChannelHeader_t);
	ServiceChannel.pResponseValues := ADR(ResponseData) + SIZEOF(ServiceChannelHeader_t);
	RequestHeader ACCESS ADR(RequestData);
	ResponseHeader ACCESS ADR(ResponseData);

END_ACTION

(* Sequence service channel execution *)
ACTION SequenceServiceChannelExecution:

	IF ServiceChannel.state = scSTATE_RECV AND RequestHeader.sequence <> ResponseHeader.sequence THEN
		ServiceChannel.requestSequence := RequestHeader.sequence;
		ServiceChannel.state := scSTATE_EXEC;

	ELSIF ServiceChannel.state = scSTATE_EXEC OR ServiceChannel.state = scSTATE_WAIT THEN
		SuperTrakServiceChannel(ServiceChannel);

	ELSIF ServiceChannel.state = scSTATE_SEND THEN
		LogServiceChannelRequest;
		ServiceChannel.state := scSTATE_RECV;
	END_IF

END_ACTION

(* Log request data when service channel request is sent *)
ACTION LogServiceChannelRequest:

	// Read Section Count 1080
	// Read System Name 1053
	// Read Enable Signal Source 1057
	// Write PLC Interface Options 1430
	// Write PLC Interface Section Count 1432
	// Write PLC Interface Target Count 1434
	// Write PLC Interface Command Count 1436
	// Write Parameter Save Function 971

	Values.i[0] := RequestHeader.task;
	Values.i[1] := RequestHeader.param;
	Values.i[2] := RequestHeader.section;
	Values.i[3] := RequestHeader.count;
	UserLogAdvanced(USERLOG_SEVERITY_INFORMATION, 100, 'Service Channel Request: Task %i, Parameter %i, Section %i, Count %i', Values);

END_ACTION

(* Call service channel address and sequence actions *)
ACTION ProcessServiceChannel:

	AddressServiceChannel;
	SequenceServiceChannelExecution;

END_ACTION
```

#### Log.var - not listed in the package file held
```iecst
VAR
	PreviousServiceChannelState : USINT; (*Montior for change in service channel processing states*)
	Values : UserLogFormatType; (*Runtime values for formatted log messages*)
END_VAR
```

### Package Logical/Source/MachineMgr/STMgr/STSystem - 1100 StCom system control

### Program Logical/Source/MachineMgr/STMgr/STSystem/STSystem

#### Types.typ
```iecst
TYPE
	StateEnum :
		(
		STATE_OFF, (*No action, wait for start*)
		STATE_INITIALIZE, (*Enable StControl function block*)
		STATE_IDLE, (*No action, wait for run*)
		STATE_STARTING, (*Enable all sections*)
		STATE_EXECUTE, (*Running, wait for stop*)
		STATE_STOPPING, (*Disable all sections*)
		STATE_ERROR, (*An error occurred*)
		STATE_CLEARING (*Reset error*)
		);
	AlarmEnum :
		(
		ALARM_COMMAND_TIMEOUT,
		ALARM_STCONTROL_ERROR
		);
END_TYPE
```

#### Variables.var
```iecst
(*Control*)
VAR
	State : StateEnum;
	Interface : STSystemInterfaceType;
END_VAR
(*Function blocks*)
VAR
	EnableTrigger : R_TRIG;
	RunTrigger : R_TRIG;
	ResetTrigger : R_TRIG;
	ControlSystem : StControl;
	SystemParameters : StControlParType;
	Timeout : TON;
END_VAR
(*Data*)
VAR
	SectionStatus : REFERENCE TO USINT;
	PLCInterfaceConfiguration : SuperTrakControlIfConfig_t;
	Index : UINT;
END_VAR
```

#### Diagram.md
~~~~markdown
Built with [Mermaid](https://mermaid.live/).

```mermaid
---
title: STSystem
---
stateDiagram
    classDef actingState stroke-dasharray:5
    state error_state <<join>>
    state execute_state <<join>>
    state stopped_state <<join>>

    [*] --> OFF
    OFF --> INITIALIZE : StartTrigger
    INITIALIZE --> error_state
    INITIALIZE --> IDLE : Active
    IDLE --> error_state
    IDLE --> execute_state
    IDLE --> STARTING : RunTrigger
    STARTING --> error_state
    STARTING --> execute_state
    EXECUTE --> error_state
    EXECUTE --> STOPPING: Stop
    EXECUTE --> stopped_state
    STOPPING --> stopped_state
    ERROR --> CLEARING: ResetTrigger
    CLEARING --> [*]

    error_state --> ERROR: Error
    execute_state --> EXECUTE: SectionsEnabled
    stopped_state --> IDLE: SectionsDisabled

    class INITIALIZE, STARTING, STOPPING, CLEARING actingState
```
~~~~

#### Main.st
```iecst
PROGRAM _INIT

	SystemParameters.NrOfCommands := 24;
	SystemParameters.NrOfSections := 4;
	SystemParameters.NrOfTargets := 4;
	SystemParameters.NrOfPallets := 4;

	Timeout.PT := T#500ms;

END_PROGRAM

PROGRAM _CYCLIC

	// Read global inputs
	Interface.Cmd := gSTSystem.Cmd;

	// State control
	CASE State OF
		STATE_OFF:
			IF EnableTrigger.Q THEN
				State := STATE_INITIALIZE;
			END_IF

		STATE_INITIALIZE;
			// Enable once and never disabled
            ControlSystem.Enable := TRUE;

			IF ControlSystem.Active THEN
				State := STATE_IDLE;

			ELSIF ControlSystem.Error THEN
				Interface.Status.ErrorID := ControlSystem.StatusID;
				State := STATE_ERROR;

			ELSIF Timeout.Q THEN
				Interface.Status.ErrorID := -1;
				State := STATE_ERROR;
            END_IF

		STATE_IDLE:
			IF ControlSystem.SectionsEnabled THEN
				UserLogBasic(USERLOG_SEVERITY_WARNING, 1102, 'Sections enabled by alternative source');
				State := STATE_EXECUTE;

			ELSIF RunTrigger.Q THEN
				State := STATE_STARTING;

			ELSIF ControlSystem.Error THEN
				Interface.Status.ErrorID := ControlSystem.StatusID;
				State := STATE_ERROR;
			END_IF

        STATE_STARTING:
            ControlSystem.EnableAllSections := TRUE;

            IF ControlSystem.SectionsEnabled THEN
                State := STATE_EXECUTE;

			ELSIF ControlSystem.Error THEN
				Interface.Status.ErrorID := ControlSystem.StatusID;
				State := STATE_ERROR;

			ELSIF Timeout.Q THEN
				Interface.Status.ErrorID := -1;
				State := STATE_ERROR;
			END_IF

		STATE_EXECUTE:
			IF Interface.Info.SectionsDisabled THEN
				UserLogBasic(USERLOG_SEVERITY_WARNING, 1104, 'Sections disabled by alternative source');
				ControlSystem.EnableAllSections := FALSE;
				State := STATE_IDLE;

			ELSIF Interface.Cmd.Stop THEN
				State := STATE_STOPPING;

			ELSIF ControlSystem.Error THEN
				Interface.Status.ErrorID := ControlSystem.StatusID;
				State := STATE_ERROR;
			END_IF

		STATE_STOPPING:
			ControlSystem.EnableAllSections := FALSE;

			IF Interface.Info.SectionsDisabled THEN
				State := STATE_IDLE;

			ELSIF ControlSystem.Error THEN
				Interface.Status.ErrorID := ControlSystem.StatusID;
				State := STATE_ERROR;

			ELSIF Timeout.Q THEN
				Interface.Status.ErrorID := -1;
				State := STATE_ERROR;
			END_IF

		STATE_ERROR:
			ControlSystem.EnableAllSections := FALSE;

			IF ResetTrigger.Q THEN
				State := STATE_CLEARING;
			END_IF

		STATE_CLEARING:
			ControlSystem.ErrorReset := TRUE;
			Interface.Status.ErrorID := 0;

			IF ControlSystem.Error = FALSE THEN
				ControlSystem.ErrorReset := FALSE;
				State := STATE_OFF;

			ELSIF Timeout.Q THEN
				Interface.Status.ErrorID := -1;
				State := STATE_ERROR;
			END_IF
	END_CASE

    // Call function blocks
    ControlSystem.StCtrlData := gSTCyclicRef.ControlDataAddress;
	ControlSystem.StCtrlDataSize := gSTCyclicRef.ControlDataSize;
	ControlSystem.StStatData := gSTCyclicRef.StatusDataAddress;
	ControlSystem.StStatDataSize := gSTCyclicRef.StatusDataSize;
	ControlSystem.StServChRequestData := gSTCyclicRef.RequestDataAddress;
	ControlSystem.StServChRequestDataSize := gSTCyclicRef.RequestDataSize;
	ControlSystem.StServChResponseData := gSTCyclicRef.ResponseDataAddress;
	ControlSystem.StServChResponseDataSize := gSTCyclicRef.ResponseDataSize;
	ControlSystem.StLink := ADR(gSTSystemLink);
	ControlSystem.Parameters := ADR(SystemParameters);
	ControlSystem();

	EnableTrigger.CLK := Interface.Cmd.Enable;
	EnableTrigger();
	RunTrigger.CLK := Interface.Cmd.Run;
	RunTrigger();
	ResetTrigger.CLK := Interface.Cmd.Reset;
	ResetTrigger();

	Timeout.IN := Interface.Status.Busy;
	Timeout();

	// Process outputs
	CollectSectionStatuses;
	Interface.Info.WarningPresent := ControlSystem.Info.SuperTrak.SystemWarningActive;
	Interface.Info.Warnings := ControlSystem.Info.SuperTrak.SystemWarningBits;
	Interface.Info.FaultPresent := ControlSystem.Info.SuperTrak.SystemFaultActive;
	Interface.Info.Faults := ControlSystem.Info.SuperTrak.SystemFaultBits;

    // Set status
    Interface.Status.Active := ControlSystem.Active;
	Interface.Status.Busy := State = STATE_INITIALIZE OR
							State = STATE_STARTING OR
							State = STATE_STOPPING OR
							State = STATE_CLEARING;
	Interface.Status.Ready := Interface.Cmd.Stop = FALSE AND State = STATE_IDLE;
	Interface.Status.Running := State = STATE_EXECUTE;
	Interface.Status.Stopped := Interface.Cmd.Stop AND State = STATE_IDLE;
	Interface.Status.Error := State = STATE_ERROR;

	// Write global outputs
	gSTSystem.Status := Interface.Status;
	gSTSystem.Info := Interface.Info;

END_PROGRAM

PROGRAM _EXIT

END_PROGRAM
```

### Package Logical/Source/MachineMgr/STMgr/STSection - StCom section control

### STSection.var
```iecst
VAR CONSTANT
	ST_SECTION_MAX : USINT := 4;
END_VAR
VAR
	gSTSection : STSectionInterfaceType;
END_VAR
```

### Program Logical/Source/MachineMgr/STMgr/STSection/STSection

#### Main.st
```iecst
PROGRAM _INIT

END_PROGRAM

PROGRAM _CYCLIC

    // Read global inputs
    Interface.Cmd := gSTSection.Cmd;

	// Initialize common statuses, assume true/false then disqualify
	Interface.Status.Active := TRUE;
	Interface.Status.Error := FALSE;

	FOR Index := 1 TO ST_SECTION_MAX DO
		ControlSection[Index].StLink := ADR(gSTSystemLink);
		ControlSection[Index].Section := Index;
		// There are no function block parameters, use common address
		ControlSection[Index].Parameters := ADR(SectionParameters);
		// Enable all function blocks
		ControlSection[Index].Enable := Interface.Cmd.Enable;
		// Enable each section
		ControlSection[Index].EnableSection := Interface.Cmd.EnableSection[Index] AND ControlSection[Index].MotorPowerOn AND NOT ControlSection[Index].Error;
		// Reset all function blocks
		ControlSection[Index].ErrorReset := Interface.Cmd.Reset;
		ControlSection[Index]();

		// All sections must be active
		IF ControlSection[Index].Active = FALSE THEN
			Interface.Status.Active := FALSE;
		END_IF
		// Error if any section has error
		IF ControlSection[Index].Error THEN
            Interface.Status.Error := TRUE;
            Interface.Status.StatusID := ControlSection[Index].StatusID;
		END_IF
		Interface.Status.SectionEnabled[Index] := ControlSection[Index].SectionEnabled;
    END_FOR

    // Write global outputs
    gSTSection.Status := Interface.Status;

END_PROGRAM

PROGRAM _EXIT

END_PROGRAM
```

### Package Logical/Source/STMgr - SuperTrak manager

### SuperTrak.typ - Global SuperTrak types
```iecst
(***************************************************************************************
 * Global SuperTrak data types
 *
 * These structures allow any program (task) to interface with the SuperTrak (ST) tasks
 *
 * File: SuperTrak.typ
 * Created: 2024-08-15
 *
 * Authors:
 *  Marcus Mangel, B&R Industrial Automation
 *
****************************************************************************************)

TYPE
    SuperTrak_type :     STRUCT  (*Main SuperTrak command/parameter/status structure*)
        System : STSystemInterfaceType; (*SuperTrak System interface*)
        Sections : STSectionInterfaceType; (*SuperTrak Section interface*)
        Target : ARRAY[1..ST_TARGET_MAX]OF STTargetInterfaceType; (*SuperTrak Targets interface*)
        Shuttle : ARRAY[1..ST_SHUTTLE_MAX]OF STShuttleInterfaceType; (*SuperTrak Shuttles interface*)
    END_STRUCT;
    STReleaseCommandType :     STRUCT  (*Release (target and shuttle) command structure*)
        ReleaseToTarget : BOOL; (*Release shuttle to target. Configure destination, direction, velocity, and acceleration.*)
        ReleaseToOffset : BOOL; (*Release shuttle to target with a configured offset. Configure destination, direction, velocity, acceleration, and offset.*)
        IncrementOffset : BOOL; (*Increment the shuttle offset. Configure velocity, acceleration, and incremental distance.*)
    END_STRUCT;
    STReleaseParameterType :     STRUCT  (*Release (target and shuttle) parameter structure*)
        Velocity : REAL; (*[mm/s] Set velocity of release movement (10..4000)*)
        Acceleration : REAL; (*[m/s^2] Set acceleration of release movement (1..60)*)
        Direction : StParamAdvReleaseConfigDirEnum; (*Direction of release movement 0: left (CW) 1: right (CCW)*)
        DestinationTarget : USINT := 1; (*1..254 Destination target, target configured in TrackMaster, 255 identified for expert mode*)
        TargetOffset : REAL; (*[mm] Absolute position offset relative to destination target (-500..500)*)
        IncrementalOffset : REAL; (*[mm] Increment current accumulated offset of current destination target (-500..500)*)
    END_STRUCT;
END_TYPE
```

### SuperTrak.var - Global SuperTrak variables
```iecst
(***************************************************************************************
 * Global SuperTrak variables
 *
 * These variables allow any program (task) to interface with the SuperTrak (ST) tasks
 *
 * File: SuperTrak.var
 * Created: 2024-08-15
 *
 * Authors:
 *  Marcus Mangel, B&R Industrial Automation
 *
****************************************************************************************)
(*SuperTrak Structure*)
VAR
    gSuperTrak : SuperTrak_type; (*Main SuperTrak command/parameter/status structure*)
END_VAR
(*Array Size Constants*)
VAR CONSTANT
    ST_SECTION_MAX : USINT := 8; (*Maximum Section number (change if adding sections)*)
    ST_TARGET_MAX : USINT := 32; (*MUST BE DIVISIBLE BY 4. Maximum Target number (change if adding targets). Should be > actual number of targets*)
    ST_SHUTTLE_MAX : USINT := 30; (*Maximum Shuttle number (change if adding shuttles)*)
END_VAR
(*Conversion*)
VAR CONSTANT
    METERS_TO_MILLIMETERS : REAL := 1000.0; (*Convert acceleration values from m/s^2 to mm/s^2*)
END_VAR
```

### Package Logical/Source/STMgr/STCyclic - SuperTrak cyclic update

### STCyclic.typ - Global types
```iecst
(***************************************************************************************
 * Global STCyclic data types
 *
 * These SuperTrak Cyclic program structures must be accessed by other tasks
 *
 * File: STCyclic.typ
 * Created: 2024-01-12
 *
 * Authors:
 *  Tyler Matijevich, B&R Industrial Automation
 *
****************************************************************************************)

TYPE
	STCyclicRefType : 	STRUCT  (*SuperTrak cyclically referenced data*)
		ControlDataAddress : UDINT; (*Pointer to array of USINT*)
		ControlDataSize : UDINT; (*[bytes] Size of Control Data array*)
		StatusDataAddress : UDINT; (*Pointer to array of USINT*)
		StatusDataSize : UDINT; (*[bytes] Size of Status Data array*)
		RequestDataAddress : UDINT; (*Pointer to array of USINT for service channel request data *)
		RequestDataSize : UDINT; (*[bytes] Size of Request Data array*)
		ResponseDataAddress : UDINT; (*Pointer to array of USINT for service channel response data *)
		ResponseDataSize : UDINT; (*[bytes] Size of Response Data array*)
	END_STRUCT;
END_TYPE
```

### STCyclic.var - Global variables
```iecst
(***************************************************************************************
 * Global STCyclic variables
 *
 * These SuperTrak Cyclic program variables must be accessed by other tasks
 *
 * File: STCyclic.var
 * Created: 2024-01-12
 *
 * Authors:
 *  Tyler Matijevich, B&R Industrial Automation
 *
***************************************************************************************)
VAR
	gSTCyclicRef : STCyclicRefType; (*SuperTrak cyclically referenced data*)
END_VAR
```

### Program Logical/Source/STMgr/STCyclic/STCyclic (IEC) - SuperTrak cyclic update

#### Main.st - Init, cyclic, exit code
```iecst
(***************************************************************************************
 * STCyclic task
 *
 * This task calls all of the functions cyclically necessary to run a SuperTrak
 * IMPORTANT: This task must be called in Cyclic #1. Cycle time: 800us, Tolerance: 0us.
 * THIS IS A REQUIREMENT TO USE SUPERTRAK.
 *
 * To change the location of the SuperTrak configuration (.dat) files, modify
 * the path used by the SuperTrakInit function in the INIT program.
 *
 * File: STCyclic.st
 * Created: 2024-01-12
 *
 * Authors:
 *  Tyler Matijevich, B&R Industrial Automation
 *
***************************************************************************************)

PROGRAM _INIT

    CheckTaskClass; // Check that task is running in 800us task class

	// Set Config Path automatically for simulation
	ConfigPath:= '/DEVICE=USER_PATH\SuperTrak\';

	// Initialize SuperTrak
	SuperTrakInit(ConfigPath, '127.0.0.1', 'IF3,IF4,IF5,IF6');

	InitializeControlInterface;

    DeConfigureAllowSectionEnableInputs;

END_PROGRAM

PROGRAM _CYCLIC

	// Data addresses for PLC control interface
    AddressControlInterface;

    // Overwrite StCom data to clear System and Section Faults
    ResetControlLevelFaults;

	// StCom input data
    SuperTrakProcessControl(0, InterfaceParameters);

	// SuperTrak cyclic update
	SuperTrakCyclic1();

	// StCom output data
	SuperTrakProcessStatus(0, InterfaceParameters);

	// StCom reference
	ReferenceCyclicData;

END_PROGRAM

PROGRAM _EXIT

	SuperTrakExit();

END_PROGRAM
```

#### Interface.var - Control interface variables for PLC communication
```iecst
(***************************************************************************************
 * STCyclic task local Interface variables
 *
 * These variables are local to the STCyclic task and are used for
 * the SuperTrak Control and Status interfaces
 *
 * File: STCyclic/Interface.var
 * Created: 2024-01-12
 *
 * Authors:
 *  Tyler Matijevich, B&R Industrial Automation
 *
***************************************************************************************)
VAR
    ControlInterfaceRevision : UINT; (*Revision number 0 required for StCom*)
    ControlData : ARRAY[0..499] OF USINT := [500(0)]; (*Raw input data to control interface*)
    StatusData : ARRAY[0..499] OF USINT := [500(0)]; (*Raw output data from control interface*)
    InterfaceParameters : SuperTrakControlInterface_t; (*Control interface parameters*)
    UserLogArguments : UserLogFormatType; (*Arguments used in Logger messages (UserLog library)*)
    fb_RTInfo : RTInfo; (*Gets information about the current runtime task*)
    ConfigPath : STRING[80]; (*Location of TrakMaster .dat files*)
    PLCInterfaceConfiguration : SuperTrakControlIfConfig_t; (*PLC Interface Configuration, used to access configured section count*)
    SystemControl : REFERENCE TO USINT; (*System Control data. Used to write Fault Reset bit*)
    SectionControl : REFERENCE TO USINT; (*Individual Section Control data. Used to write Fault Reset bit*)
    Index : UINT; (*FOR loop index*)
END_VAR
```

#### Interface.st - Control interface actions for PLC communication
```iecst
(***************************************************************************************
 * STCyclic task Interface actions
 *
 * These Actions can be run only by the STCyclic task and relate to the
 * SuperTrak Control and Status interfaces
 *
 * File: STCyclic/Interface.st
 * Created: 2024-01-12
 *
 * Authors:
 *  Tyler Matijevich, B&R Industrial Automation
 *  Marcus Mangel, B&R Industrial Automation
 *
***************************************************************************************)

(* Check that task is running in 800us task class and log if not *)
ACTION CheckTaskClass:

    fb_RTInfo(enable := TRUE);
    IF fb_RTInfo.cycle_time <> 800 OR fb_RTInfo.task_class <> 1 THEN
        brsmemset(ADR(UserLogArguments), 0, SIZEOF(UserLogArguments));
        UserLogEventText('$$arlogusr', -536869912, 0, '', '', UserLogArguments);
    END_IF;

END_ACTION

(* Assign revision, connection type, and size of control interface data *)
ACTION InitializeControlInterface:

	// Revision 0 required by StCom
	ControlInterfaceRevision := 0;
	SuperTrakServChanWrite(0, stPAR_PLC_IF_REVISION, 0, 1,
		ADR(ControlInterfaceRevision), SIZEOF(ControlInterfaceRevision));

	// Parameters used in SuperTrak ProcessControl and ProcessStatus functions
	InterfaceParameters.connectionType := stCONNECTION_LOCAL;
	InterfaceParameters.controlSize := SIZEOF(ControlData);
	InterfaceParameters.statusSize := SIZEOF(StatusData);

END_ACTION

(* Assign addresses of control interface data *)
ACTION AddressControlInterface:

	// Parameters used in SuperTrak ProcessControl and ProcessStatus functions
    InterfaceParameters.pControl := ADR(ControlData);
    InterfaceParameters.pStatus := ADR(StatusData);

END_ACTION

(* Reset Faults and Warnkngs for all Sections as well as the System *)
// This functionality is not implemented by StCom and so it must be done from the
// cyclic control layer. The same functionality can be achieved with the Clear Faults
// button in TrakMaster.
ACTION ResetControlLevelFaults:

    // Read PLC interface configuration (counts and offsets)
    SuperTrakGetControlIfConfig(0, PLCInterfaceConfiguration);

    // Reset System level faults
    SystemControl ACCESS ADR(ControlData) + PLCInterfaceConfiguration.systemControlOffset;
    SystemControl.7 := gSuperTrak.System.Cmd.Reset; // Bit 7 is Acknowledge Faults. See TrakMaster Help.
    // !! The data at this address is also modified by StCom. Do not modify any other bits !!

    // Stop here if there are no sections configured
    IF PLCInterfaceConfiguration.sectionCount = 0 THEN
        RETURN;
    END_IF

    // Loop through every configured section
    FOR Index := 0 TO PLCInterfaceConfiguration.sectionCount - 1 DO
        SectionControl ACCESS ADR(ControlData) + PLCInterfaceConfiguration.sectionControlOffset + Index;
        SectionControl.7 := gSuperTrak.System.Cmd.Reset; // Bit 7 is Acknowledge Faults. See TrakMaster Help.
        // !! The data at this address is also modified by StCom. Do not modify any other bits !!
    END_FOR

END_ACTION
```

#### Service.var - Service channel variables
```iecst
(***************************************************************************************
 * STCyclic task local Service variables
 *
 * These variables are local to the STCyclic task and are used for
 * SuperTrak Service Channel requests/responses
 *
 * File: STCyclic/Service.var
 * Created: 2024-01-12
 *
 * Authors:
 *  Tyler Matijevich, B&R Industrial Automation
 *
***************************************************************************************)
VAR
	RequestData : ARRAY[0..127] OF USINT := [128(0)]; (*Raw service channel input data*)
	ResponseData : ARRAY[0..127] OF USINT := [128(0)]; (*Raw service channel output data*)
END_VAR
(*Configure Digital Inputs*)
VAR
	DigtalInputFunctions : ARRAY[0..7] OF UINT; (*Each array element corresponds to a Digital Input in Trakmaster*)
	InputParameterDataLength : UDINT; (*Data length for Digital Input parameter*)
	InputCount : UINT; (*Number of digital inputs available*)
	InputIndex : USINT; (*FOR Loop index*)
	InputConfigChanged : BOOL; (*Flag that input configuration needs to be written back*)
END_VAR
```

#### Service.st - Service channel actions
```iecst
(***************************************************************************************
 * STCyclic task Service actions
 *
 * These Actions can be run only by the STCyclic task and relate to the
 * SuperTrak Service Channel
 *
 * File: STCyclic/Service.st
 * Created: 2024-01-12
 *
 * Authors:
 *  Tyler Matijevich, B&R Industrial Automation
 *
***************************************************************************************)

(* De-Configure any "Allow Section Enable" inputs *)
ACTION DeConfigureAllowSectionEnableInputs:
    InputConfigChanged := FALSE;

    // Data parameters occupy parameter numbers starting at 1024
    // To obtain information about data parameter K, specify index K - 1024 when reading the Data Parameter Information parameters
    SuperTrakServChanRead(0, stPAR_PARAM_ARRAY_LENGTH, stPAR_DIGITAL_INPUT_FUNCTION - 1024, 1, ADR(InputParameterDataLength), SIZEOF(InputParameterDataLength));

    // Number of inputs is lesser of (data array size, size of data buffer elements)
    InputCount := MIN(UDINT_TO_UINT(InputParameterDataLength), SIZEOF(DigtalInputFunctions)/SIZEOF(DigtalInputFunctions[0]));
    SuperTrakServChanRead(0, stPAR_DIGITAL_INPUT_FUNCTION, 0, InputCount, ADR(DigtalInputFunctions), SIZEOF(DigtalInputFunctions));

    FOR InputIndex := 0 TO 7 DO
        IF DigtalInputFunctions[InputIndex] = 25 THEN // 25 means input is configured as Allow Section Enable
            DigtalInputFunctions[InputIndex] := 0; // 0 means Not Configured
            InputConfigChanged := TRUE;
        END_IF;
    END_FOR;

    IF InputConfigChanged THEN
        SuperTrakServChanWrite(0, stPAR_DIGITAL_INPUT_FUNCTION, 0, InputCount, ADR(DigtalInputFunctions), SIZEOF(DigtalInputFunctions));
    END_IF;

END_ACTION
```

#### Reference.st - Reference control interface and service channel for StCom
```iecst
(***************************************************************************************
 * STCyclic task Cyclic Reference actions
 *
 * These Actions can be run only by the STCyclic task and relate to the
 * SuperTrak cyclic reference variable used by StCom function blocks
 *
 * File: STCyclic/Reference.st
 * Created: 2024-01-12
 *
 * Authors:
 *  Tyler Matijevich, B&R Industrial Automation
 *
***************************************************************************************)

(* Reference control interface and service channel data *)
ACTION ReferenceCyclicData:

	gSTCyclicRef.ControlDataAddress := ADR(ControlData);
	gSTCyclicRef.ControlDataSize := SIZEOF(ControlData);
	gSTCyclicRef.StatusDataAddress := ADR(StatusData);
	gSTCyclicRef.StatusDataSize := SIZEOF(StatusData);
	gSTCyclicRef.RequestDataAddress := ADR(RequestData);
	gSTCyclicRef.RequestDataSize := SIZEOF(RequestData);
	gSTCyclicRef.ResponseDataAddress := ADR(ResponseData);
	gSTCyclicRef.ResponseDataSize := SIZEOF(ResponseData);

END_ACTION
```

### Package Logical/Source/STMgr/STSystem - StCom system control

### STSystem.typ - Global types
```iecst
(***************************************************************************************
 * Global STSystem data types
 *
 * These structures allow any program (task) to interface with the STSystem task
 *
 * File: STSystem.typ
 * Created: 2024-08-15
 *
 * Authors:
 *  Marcus Mangel, B&R Industrial Automation
 *
****************************************************************************************)

TYPE
	STSystemInterfaceType : 	STRUCT  (*Program interface*)
		Cmd : STSystemInterfaceCmdType; (*System commands*)
		Par : STSystemInterfaceParType; (*System parameters*)
		Status : STSystemInterfaceStatusType; (*Status of the System interface*)
		Info : STSystemInterfaceInfoType; (*System information*)
	END_STRUCT;
	STSystemInterfaceCmdType : 	STRUCT  (*Interface commands*)
		PowerAllSections : BOOL; (*Run the SuperTrak via System Control (enable all sections)*)
		Reset : BOOL; (*Error Reset*)
	END_STRUCT;
	STSystemInterfaceParType : 	STRUCT  (*Interface parameters*)
		GlobalDirection : UINT := 1; (*Define global direction 0: left (CW) 1: right (CCW)*)
	END_STRUCT;
	STSystemInterfaceStatusType : 	STRUCT  (*Interface command response*)
		Active : BOOL; (*Control function block is Active*)
		Busy : BOOL; (*Interface is processing a command*)
		Ready : BOOL; (*Interface is ready for commands*)
		PowerOn : BOOL; (*Sections are enabled*)
		Error : BOOL; (*There is an active error in the task*)
		ErrorID : DINT; (*ID of the active error*)
	END_STRUCT;
	STSystemInterfaceInfoType : 	STRUCT  (*Interface information*)
		WarningPresent : BOOL; (*One or more system warnings are active*)
		Warnings : UDINT; (*System warning bits*)
		FaultPresent : BOOL; (*One or more system faults are active*)
		Faults : UDINT; (*System fault bits*)
		SectionCount : UINT; (*Number of configured sections (only read once on control enable)*)
		ShuttleCount : UINT; (*Number of shuttles currently on the system (read cyclically)*)
		SectionsEnabled : BOOL; (*All sections enabled*)
		SectionsDisabled : BOOL; (*All sections disabled*)
	END_STRUCT;
END_TYPE
```

### STSystem.var - Global variables
```iecst
(***************************************************************************************
 * Global STSystem variables
 *
 * These SuperTrak System variables must be accessed by other tasks
 *
 * File: STCyclic.var
 * Created: 2024-01-12
 *
 * Authors:
 *  Tyler Matijevich, B&R Industrial Automation
 *
***************************************************************************************)
VAR
	gSTSystemLink : StLinkType; (*StCom SuperTrak cyclic reference*)
END_VAR
```

### Program Logical/Source/STMgr/STSystem/STSystem (IEC) - StCom system control

#### Main.st - Init, cyclic, exit code
```iecst
(***************************************************************************************
 * STSystem task
 *
 * This task provides a state machine for enabling/disabling the SuperTrak system.
 * This task should be controlled by the Main task via gSuperTrak.System.
 *
 * If adding sections, targets, or shuttles, double check the assigned values
 * of the ST_XX_MAX constants.
 *
 * File: STSystem.st
 * Created: 2024-08-15
 *
 * Authors:
 *  Marcus Mangel, B&R Industrial Automation
 *  Tyler Matijevich, B&R Industrial Automation
 *
***************************************************************************************)

PROGRAM _INIT

    // Set "number of" parameters to be size of their respective arrays
    // If more Sections, Pallets, or Targets are added these constants must be updated.
    // But follow the instructions in the constant's description!
	SystemParameters.NrOfCommands := ST_COMMAND_MAX;
	SystemParameters.NrOfSections := ST_SECTION_MAX;
	SystemParameters.NrOfTargets := ST_TARGET_MAX; // This must be divisible by 4 and must be at least 1 more than the actual number of Targets
	SystemParameters.NrOfPallets := ST_SHUTTLE_MAX;

	Timeout.PT := T#5000ms;

END_PROGRAM

PROGRAM _CYCLIC

	// Read global inputs
    Interface.Cmd := gSuperTrak.System.Cmd;

    // State control
    CASE State OF
        STATE_INITIALIZE:
            // Enable once and never disabled
            ControlSystem.Enable := TRUE;

            IF ControlSystem.Active THEN
                brsmemset(ADR(UserLogArguments), 0, SIZEOF(UserLogArguments));
                UserLogArguments.i[0] := SystemParameters.NrOfSections;
                UserLogArguments.i[1] := SystemParameters.NrOfTargets;
                UserLogArguments.i[2] := SystemParameters.NrOfPallets;
                UserLogCustom('$$arlogusr', USERLOG_SEVERITY_INFORMATION, 1, 31, 0, '', 'StControl Active. Max: Sections %i, Targets %i, Shuttles %i', UserLogArguments);
                State := STATE_IDLE;

            ELSIF ControlSystem.Error THEN
                Interface.Status.ErrorID := ControlSystem.StatusID;
                brsmemset(ADR(UserLogArguments), 0, SIZEOF(UserLogArguments));
                UserLogArguments.i[0] := ControlSystem.StatusID;
                UserLogEventText('$$arlogusr', -536869902, 0, '', '%i', UserLogArguments);
                State := STATE_ERROR;

            ELSIF Timeout.Q THEN
                Interface.Status.ErrorID := -1;
                brsmemset(ADR(UserLogArguments), 0, SIZEOF(UserLogArguments));
                UserLogEventText('$$arlogusr', -536868912, 0, '', '', UserLogArguments);
                State := STATE_ERROR;
            END_IF

		STATE_IDLE:
            IF ControlSystem.SectionsEnabled THEN
                brsmemset(ADR(UserLogArguments), 0, SIZEOF(UserLogArguments));
                UserLogEventText('$$arlogusr', -1610609736, 0, '', '', UserLogArguments);
                State := STATE_EXECUTE;

            ELSIF RunTrigger.Q THEN
                State := STATE_STARTING;

            ELSIF ControlSystem.Error THEN
                Interface.Status.ErrorID := ControlSystem.StatusID;
                brsmemset(ADR(UserLogArguments), 0, SIZEOF(UserLogArguments));
                UserLogArguments.i[0] := ControlSystem.StatusID;
                UserLogEventText('$$arlogusr', -536869902, 0, '', '%i', UserLogArguments);
                State := STATE_ERROR;
            END_IF

        STATE_STARTING:
            ControlSystem.EnableAllSections := TRUE;

            IF ControlSystem.SectionsEnabled THEN
                brsmemset(ADR(UserLogArguments), 0, SIZEOF(UserLogArguments));
                UserLogCustom('$$arlogusr', USERLOG_SEVERITY_INFORMATION, 1, 32, 0, '', 'StControl: All Sections Enabled', UserLogArguments);
                State := STATE_EXECUTE;

            ELSIF ControlSystem.Error THEN
                Interface.Status.ErrorID := ControlSystem.StatusID;
                brsmemset(ADR(UserLogArguments), 0, SIZEOF(UserLogArguments));
                UserLogArguments.i[0] := ControlSystem.StatusID;
                UserLogEventText('$$arlogusr', -536869902, 0, '', '%i', UserLogArguments);
                State := STATE_ERROR;

            ELSIF Timeout.Q THEN
                Interface.Status.ErrorID := -1;
                brsmemset(ADR(UserLogArguments), 0, SIZEOF(UserLogArguments));
                UserLogEventText('$$arlogusr', -536868911, 0, '', '', UserLogArguments);
                State := STATE_ERROR;
            END_IF

        STATE_EXECUTE:
            IF Interface.Info.SectionsDisabled THEN
                brsmemset(ADR(UserLogArguments), 0, SIZEOF(UserLogArguments));
                UserLogEventText('$$arlogusr', -1610609735, 0, '', '', UserLogArguments);
                ControlSystem.EnableAllSections := FALSE;
                State := STATE_IDLE;

            ELSIF NOT Interface.Cmd.PowerAllSections THEN
                State := STATE_STOPPING;

            ELSIF ControlSystem.Error THEN
                Interface.Status.ErrorID := ControlSystem.StatusID;
                brsmemset(ADR(UserLogArguments), 0, SIZEOF(UserLogArguments));
                UserLogArguments.i[0] := ControlSystem.StatusID;
                UserLogEventText('$$arlogusr', -536869902, 0, '', '%i', UserLogArguments);
                State := STATE_ERROR;
            END_IF

        STATE_STOPPING:
            ControlSystem.EnableAllSections := FALSE;

            IF Interface.Info.SectionsDisabled THEN
                brsmemset(ADR(UserLogArguments), 0, SIZEOF(UserLogArguments));
                UserLogCustom('$$arlogusr', USERLOG_SEVERITY_INFORMATION, 1, 33, 0, '', 'StControl: All Sections Disabled', UserLogArguments);
                State := STATE_IDLE;

            ELSIF ControlSystem.Error THEN
                Interface.Status.ErrorID := ControlSystem.StatusID;
                brsmemset(ADR(UserLogArguments), 0, SIZEOF(UserLogArguments));
                UserLogArguments.i[0] := ControlSystem.StatusID;
                UserLogEventText('$$arlogusr', -536869902, 0, '', '%i', UserLogArguments);
                State := STATE_ERROR;

            ELSIF Timeout.Q THEN
                brsmemset(ADR(UserLogArguments), 0, SIZEOF(UserLogArguments));
                UserLogEventText('$$arlogusr', -536868910, 0, '', '', UserLogArguments);
                Interface.Status.ErrorID := -1;
                State := STATE_ERROR;
            END_IF

        STATE_ERROR:
            ControlSystem.EnableAllSections := FALSE;

            IF ResetTrigger.Q THEN
                State := STATE_CLEARING;
            END_IF

        STATE_CLEARING:
            ControlSystem.ErrorReset := TRUE;
            Interface.Status.ErrorID := 0;

            IF ControlSystem.Error = FALSE THEN
                ControlSystem.ErrorReset := FALSE;
                State := STATE_IDLE;

            ELSIF Timeout.Q THEN
                Interface.Status.ErrorID := -1;
                brsmemset(ADR(UserLogArguments), 0, SIZEOF(UserLogArguments));
                UserLogEventText('$$arlogusr', -536868909, 0, '', '', UserLogArguments);
                State := STATE_ERROR;
            END_IF
    END_CASE

    // Call function blocks
    ControlSystem.StCtrlData := gSTCyclicRef.ControlDataAddress;
    ControlSystem.StCtrlDataSize := gSTCyclicRef.ControlDataSize;
    ControlSystem.StStatData := gSTCyclicRef.StatusDataAddress;
    ControlSystem.StStatDataSize := gSTCyclicRef.StatusDataSize;
    ControlSystem.StServChRequestData := gSTCyclicRef.RequestDataAddress;
    ControlSystem.StServChRequestDataSize := gSTCyclicRef.RequestDataSize;
    ControlSystem.StServChResponseData := gSTCyclicRef.ResponseDataAddress;
    ControlSystem.StServChResponseDataSize := gSTCyclicRef.ResponseDataSize;
    ControlSystem.StLink := ADR(gSTSystemLink);
    ControlSystem.Parameters := ADR(SystemParameters);
    ControlSystem();

    RunTrigger.CLK := Interface.Cmd.PowerAllSections;
    RunTrigger();
    ResetTrigger.CLK := Interface.Cmd.Reset;
    ResetTrigger();

    Timeout.IN := Interface.Status.Busy;
    Timeout();

    // Process outputs
    CollectSectionStatuses;
    Interface.Info.SectionCount := ControlSystem.Info.SuperTrak.NrOfSections;
    Interface.Info.ShuttleCount := ControlSystem.Info.SuperTrak.NrOfPallets;
    Interface.Info.WarningPresent := ControlSystem.Info.SuperTrak.SystemWarningActive;
    Interface.Info.Warnings := ControlSystem.Info.SuperTrak.SystemWarningBits;
    Interface.Info.FaultPresent := ControlSystem.Info.SuperTrak.SystemFaultActive;
    Interface.Info.Faults := ControlSystem.Info.SuperTrak.SystemFaultBits;

    // Set status
    Interface.Status.Active := ControlSystem.Active;
    Interface.Status.Busy := State = STATE_INITIALIZE OR
    State = STATE_STARTING OR
    State = STATE_STOPPING OR
    State = STATE_CLEARING;
    Interface.Status.Ready := State = STATE_IDLE;
    Interface.Status.PowerOn := State = STATE_EXECUTE;
    Interface.Status.Error := State = STATE_ERROR;

    // Write global outputs
    gSuperTrak.System.Status := Interface.Status;
    gSuperTrak.System.Info := Interface.Info;

END_PROGRAM
```

#### Types.typ - Local types
```iecst
(***************************************************************************************
 * STSystem task local data types
 *
 * These structures and enumerations are local to the STSystem task
 *
 * File: STSystem/Types.typ
 * Created: 2024-08-15
 *
 * Authors:
 *  Marcus Mangel, B&R Industrial Automation
 *  Tyler Matijevich, B&R Industrial Automation
 *
***************************************************************************************)

TYPE
	StateEnum :
		( (*Program state*)
		STATE_INITIALIZE, (*Enable StControl function block*)
		STATE_IDLE, (*No action, wait for run*)
		STATE_STARTING, (*Enable all sections*)
		STATE_EXECUTE, (*Running, wait for stop*)
		STATE_STOPPING, (*Disable all sections*)
		STATE_ERROR, (*An error occurred*)
		STATE_CLEARING (*Reset error*)
		);
END_TYPE
```

#### Variables.var - Local variables
```iecst
(***************************************************************************************
 * STSystem task local variables
 *
 * These variables are local to the STSystem task
 *
 * File: STSystem/Variables.var
 * Created: 2024-08-15
 *
 * Authors:
 *  Marcus Mangel, B&R Industrial Automation
 *  Tyler Matijevich, B&R Industrial Automation
 *
***************************************************************************************)
(*Control*)
VAR
	State : StateEnum; (*Program state*)
	Interface : STSystemInterfaceType; (*Local copy of global interface*)
END_VAR
VAR CONSTANT
	ST_COMMAND_MAX : USINT := 48; (*Maximum number of commands executed simultaniously. MUST BE DIVISIBLE BY 8*)
END_VAR
(*Function blocks*)
VAR
	RunTrigger : R_TRIG; (*Rising edge trigger for Run command*)
	ResetTrigger : R_TRIG; (*Rising edge trigger for Error Reset command*)
	ControlSystem : StControl; (*StCom system control function block*)
	SystemParameters : StControlParType; (*System control parameters*)
	Timeout : TON; (*Timer to check for command timeouts*)
END_VAR
(*Data*)
VAR
	UserLogArguments : UserLogFormatType; (*Arguments used in Logger messages (UserLog library)*)
	SectionStatus : REFERENCE TO USINT; (*Status of an individual section*)
	PLCInterfaceConfiguration : SuperTrakControlIfConfig_t; (*PLC Interface Configuration, used to access configured section count*)
	Index : UINT; (*FOR loop index*)
END_VAR
```

#### Sections.st - Collect section statuses
```iecst
(***************************************************************************************
 * STSystem task Section actions
 *
 * These Actions can be run only by the STSystem task and relate to
 * individual Section control and feedback.
 *
 * File: STSystem/Sections.st
 * Created: 2024-01-12
 *
 * Authors:
 *  Tyler Matijevich, B&R Industrial Automation
 *
***************************************************************************************)

(* Collect section enable statuses *)
ACTION CollectSectionStatuses:

	Interface.Info.SectionsEnabled := ControlSystem.SectionsEnabled;

	IF ControlSystem.Active = FALSE THEN
		Interface.Info.SectionsDisabled := FALSE;
		RETURN;
	END_IF

	// Read PLC interface configuration (counts and offsets)
	SuperTrakGetControlIfConfig(0, PLCInterfaceConfiguration);
	IF PLCInterfaceConfiguration.sectionCount = 0 THEN
		RETURN;
	END_IF

	// Assume true
	Interface.Info.SectionsDisabled := TRUE;
	// Loop through every configured section
	FOR Index := 0 TO PLCInterfaceConfiguration.sectionCount - 1 DO
		SectionStatus ACCESS ControlSystem.StStatData + PLCInterfaceConfiguration.sectionStatusOffset + Index;
		// Test bit 0 if section is enabled
		IF BIT_TST(SectionStatus, 0) THEN
			Interface.Info.SectionsDisabled := FALSE;
		END_IF
	END_FOR

END_ACTION
```

### Package Logical/Source/STMgr/STSection - StCom section control

### STSection.typ - Global types
```iecst
(***************************************************************************************
 * Global STSection data types
 *
 * These structures allow any program (task) to interface with the STSection task
 *
 * File: STSection.typ
 * Created: 2024-08-15
 *
 * Authors:
 *  Marcus Mangel, B&R Industrial Automation
 *  Tyler Matijevich, B&R Industrial Automation
 *
****************************************************************************************)

TYPE
    STSectionInterfaceType :     STRUCT  (*Section control interface*)
        Cmd : STSectionInterfaceCmdType; (*Section commands*)
        Status : STSectionInterfaceStatusType; (*Section statuses*)
        Info : ARRAY[1..ST_SECTION_MAX]OF STSectionInterfaceInfoType; (*Information about each individual section*)
    END_STRUCT;
    STSectionInterfaceCmdType :     STRUCT  (*Section commands*)
        PowerSection : ARRAY[1..ST_SECTION_MAX]OF BOOL; (*Enable individual sections*)
    END_STRUCT;
    STSectionInterfaceStatusType :     STRUCT  (*Section statuses*)
        Active : BOOL; (*All section control function blocks are Active*)
        Error : BOOL; (*At least one section function block is reporting an Error*)
        StatusID : DINT; (*StatusID of section function block reporting an error*)
        SectionError : USINT; (*Section number reporting a Fault. 0 means all sections are OK*)
        SectionWarning : USINT; (*Section number reporting a Warning. 0 means all sections are OK*)
    END_STRUCT;
    STSectionInterfaceInfoType :     STRUCT  (*Information about each individual section*)
        SectionEnabled : BOOL; (*Sections that are Enabled have a TRUE value in this array*)
        UnrecognizedShuttles : BOOL; (*Detected one or more shuttles with undetermined position, jogged to locate when enabled*)
        MotorPowerOn : BOOL; (*Voltage within usage range*)
        ShuttlesRecovering : BOOL; (*Shuttles must be returned to last controlled position and/or making their initial move to load target*)
        LocatingShuttles : BOOL; (*Shuttles are automatically jogged to locate*)
        DisabledExternally : BOOL; (*Disabled due to external condition, see digital inputs*)
        WarningPresent : BOOL; (*One or more warning messages have been recorded*)
        Warnings : UDINT; (*Warning bit(s) active*)
        FaultPresent : BOOL; (*One or more fault messages have been recorded*)
        Faults : UDINT; (*Fault bit(s) active*)
    END_STRUCT;
END_TYPE
```

### Program Logical/Source/STMgr/STSection/STSection (IEC) - StCom section control

#### Variables.var
```iecst
(***************************************************************************************
 * STSection task local variables
 *
 * These variables are local to the STSection task
 *
 * File: STSection/Variables.var
 * Created: 2024-08-15
 *
 * Authors:
 *  Marcus Mangel, B&R Industrial Automation
 *  Tyler Matijevich, B&R Industrial Automation
 *
***************************************************************************************)
VAR
	Interface : STSectionInterfaceType; (*Section control interface*)
	SectionParameters : ARRAY[1..ST_SECTION_MAX] OF StSectionParType; (*Placeholder, there are no parameters for StCom's StSection function block*)
	ControlSection : ARRAY[1..ST_SECTION_MAX] OF StSection; (*Section control function block*)
	Index : USINT; (*FOR loop index*)
	UserLogArguments : UserLogFormatType; (*Arguments used in Logger messages (UserLog library)*)
	r_trig_SectionFBError : ARRAY[1..ST_SECTION_MAX] OF R_TRIG; (*Rising edge trigger for ControlSection.Error*)
	r_trig_SectionWarning : ARRAY[1..ST_SECTION_MAX] OF R_TRIG; (*Rising edge trigger for section warnings*)
	r_trig_SectionFault : ARRAY[1..ST_SECTION_MAX] OF R_TRIG; (*Rising edge trigger for section faults*)
END_VAR
```
